Universal Robots PolyScope program: DAS428_958_10_MAR_21_DAS_lado_izquierdo.urp

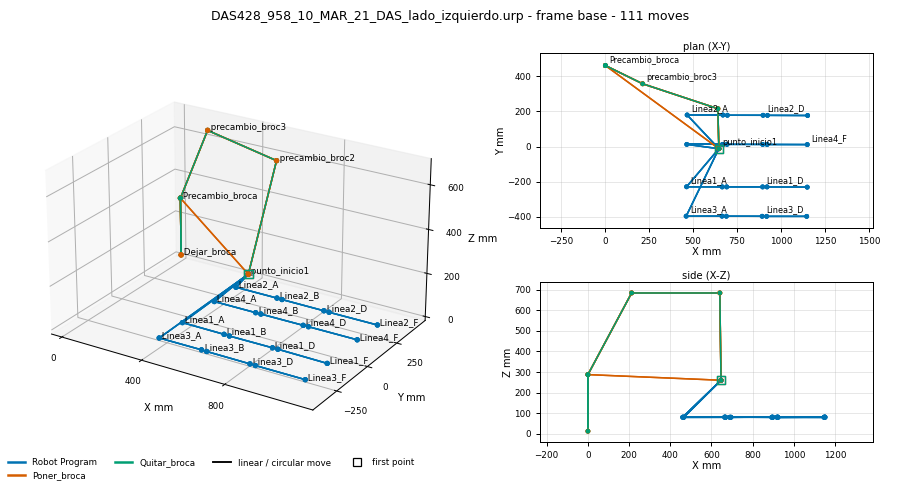
[picture p0: tool path of DAS428_958_10_MAR_21_DAS_lado_izquierdo.urp in frame base, 111 of 219 moves have a stored position in this frame; points joined in program order, loops and branches not executed]
Program DAS428_958_10_MAR_21_DAS_lado_izquierdo (installation=instalacion_derecha_10_MAR_21 directory=/programs/izquierdo createdIn=5.6.0.90886 lastSavedIn=5.6.0.90886 robotSerialNumber=20195001785)
Calibrated DH parameters: a=[0.000107, -0.568984, -0.552934, -0.00001, -0.000063, 0]; d=[0.180718, -257.998067, 200.685024, 57.48776, 0.119923, 0.115353]; alpha=[1.571119, 0.000876, -0.002498, 1.571178, -1.570523, 0]; deltaTheta=[0, -0.378191, 0.631587, -0.253396, 0, 0]
Robot Program (runOnlyOnce=false)
  Folder Variables
    bajada_broca := p[0,0,-0.008,0,0,0]
    barrenos_menos1 := 0
    barreno_actual := 0
    posicion := p[0,0,300,0,0,0]
    cambiar_broca := False
    barrenos_hechos := 0
    eje7 := 3
    Wait Sleep waitTime=0.5
  Folder Home
    Wait Sleep waitTime=0.3
    SafeHome (positionOptionType=SPEED_AND_ACCELERATION speed=1.047198 acceleration=1.396263 nextMotionTime=2)
    SuppressedNode
      MoveL speed 250 mm/s, acceleration 1200 mm/s^2 (useActiveTCP=true) feature=Base
        Waypoint home_trans: TCP in base x=-171.077 y=546.65 z=109.574 mm, rx=0.1544 ry=3.1247 rz=-0.2011 rad; joints [-91.802, -93.053, 127.954, -27.005, -275.278, -0.192] deg; TCP offset x=0.411 y=-218.298 z=37.994 mm, rx=1.558 ry=-0.1255 rz=0.1212 rad
    Wait Sleep waitTime=0.3
    iniciando_prog := True
    Call Poner_broca
  Folder Posicion2
    eje7 := 2
    Folder Broca_1
      Folder Linea1
        Folder Marcar_puntos
          MoveL speed 100 mm/s, acceleration 500 mm/s^2 (useActiveTCP=true) feature=Base
            SafeHome (positionOptionType=SPEED_AND_ACCELERATION speed=1.047198 acceleration=1.396263 nextMotionTime=2)
            Waypoint punto_inicio1: TCP in base x=646.451 y=-11.704 z=260.166 mm, rx=2.1511 ry=2.2897 rz=0 rad; joints [-205.616, -96.356, 115.768, -18.693, -308.324, -0.329] deg; TCP offset x=0.411 y=-218.298 z=37.994 mm, rx=1.558 ry=-0.1255 rz=0.1212 rad
            Waypoint Linea1_A: TCP in base x=462.97 y=-228.381 z=81.417 mm, rx=3.1274 ry=-0.0942 rz=0.0027 rad; joints [-212.166, -91.385, 132.289, -41.367, -217.89, -0.202] deg; TCP offset x=0.411 y=-218.298 z=37.994 mm, rx=1.558 ry=-0.1255 rz=0.1212 rad
            Waypoint Linea1_B: TCP in base x=665.709 y=-229.051 z=81.124 mm, rx=3.1274 ry=-0.0942 rz=0.0027 rad; joints [-202.097, -73.27, 110.874, -38.21, -207.821, -0.358] deg
            Waypoint Linea1_C: TCP in base x=691.124 y=-228.949 z=80.167 mm, rx=3.1274 ry=-0.0942 rz=0.0027 rad; joints [-201.251, -71.148, 108.001, -37.475, -206.974, -0.377] deg
            Waypoint Linea1_D: TCP in base x=895.378 y=-229.075 z=81.054 mm, rx=3.0494 ry=0.7125 rz=-0.0018 rad; joints [-199.71, -60.243, 91.126, -30.929, -235.176, -0.15] deg
            Waypoint Linea1_E: TCP in base x=920.631 y=-228.998 z=81.3 mm, rx=3.0494 ry=0.7125 rz=-0.0016 rad; joints [-199.108, -58.185, 87.734, -29.605, -234.57, -0.15] deg
            Waypoint Linea1_F: TCP in base x=1149.195 y=-230.503 z=80.116 mm, rx=3.0494 ry=0.7125 rz=-0.0018 rad; joints [-195.083, -36.259, 48.872, -12.673, -230.505, -0.164] deg
        Folder AB
          'desbaste_inicial'
          bajada_broca := p[0,0,-0.008,0,0,0]
          barrenos_menos1 := 8
          barreno_actual := 0
          Loop While (checkContinuously=false) expression=barreno_actual≤barrenos_menos1
            Folder Perforacion
              MoveL speed 100 mm/s, acceleration 500 mm/s^2 (useActiveTCP=true) feature=Base
                internos := interpolate_pose(Linea1_A, Linea1_B, barreno_actual/barrenos_menos1)
                Waypoint Waypoint (Variable): variable=internos
                'desbaste_inicial'
                bajada_broca := p[0,0,-0.008,0,0,0]
                bajada := p[0,0,0.008,0,0,0]
                MoveDirectionNode (selectedDirection=ZMinus toolParams=0.003, 0.005)
                  Until DISTANCE (allowActions=false deceleration=3 distanceNodeType=STOP) Distance=0.054; motionParameters(blendRadius=0)
                Popup Message (haltProgram=false message=punto contacto alanzdo inputType=Text)
                MoveDirectionNode (selectedDirection=ZPlus toolParams=0.003, 0.005)
                  Until DISTANCE (allowActions=false deceleration=3 distanceNodeType=STOP) Distance=0.002; motionParameters(blendRadius=0)
                Wait Sleep waitTime=0.3
                Set DigitalOutput pin=config_out[1]; digitalValue=1
                Wait Sleep waitTime=0.3
                Loop Counting (count=3) loopVariable(name=Loop_11)
                  bajar := pose_add(get_actual_tcp_pose(), bajada_broca)
                  Waypoint Waypoint (Variable): motionParameters(jointSpeed=1.047198 jointAcceleration=1.396263 cartesianSpeed=0.001 cartesianAcceleration=0.005); variable=bajar
                  subir := pose_sub(get_actual_tcp_pose(), bajada_broca)
                  Waypoint Waypoint (Variable): motionParameters(jointSpeed=1.047198 jointAcceleration=1.396263 cartesianSpeed=0.005 cartesianAcceleration=0.01); variable=subir
                  bajada_broca := pose_sub(bajada_broca, bajada)
                MoveDirectionNode (selectedDirection=ZPlus toolParams=0.03, 0.035)
                  Until DISTANCE (allowActions=false deceleration=3 distanceNodeType=STOP) Distance=0.06; motionParameters(blendRadius=0)
                Set DigitalOutput pin=config_out[1]; digitalValue=0
                barreno_actual := barreno_actual+1
                Call Quitar_broca
                Call Poner_broca
        Folder CD
          'desbaste_inicial'
          bajada_broca := p[0,0,-0.008,0,0,0]
          barrenos_menos1 := 8
          barreno_actual := 0
          Loop While (checkContinuously=false) expression=barreno_actual≤barrenos_menos1
            Folder Perforacion
              MoveL speed 100 mm/s, acceleration 500 mm/s^2 (useActiveTCP=true) feature=Base
                internos := interpolate_pose(Linea1_C, Linea1_D, barreno_actual/barrenos_menos1)
                Waypoint Waypoint (Variable): variable=internos
                'desbaste_inicial'
                bajada_broca := p[0,0,-0.008,0,0,0]
                bajada := p[0,0,0.008,0,0,0]
                MoveDirectionNode (selectedDirection=ZMinus toolParams=0.003, 0.005)
                  Until DISTANCE (allowActions=false deceleration=3 distanceNodeType=STOP) Distance=0.054; motionParameters(blendRadius=0)
                Popup Message (haltProgram=false message=punto contacto alanzdo inputType=Text)
                MoveDirectionNode (selectedDirection=ZPlus toolParams=0.003, 0.005)
                  Until DISTANCE (allowActions=false deceleration=3 distanceNodeType=STOP) Distance=0.002; motionParameters(blendRadius=0)
                Wait Sleep waitTime=0.3
                Set DigitalOutput pin=config_out[1]; digitalValue=1
                Wait Sleep waitTime=0.3
                Loop Counting (count=3) loopVariable(name=Loop_14)
                  bajar := pose_add(get_actual_tcp_pose(), bajada_broca)
                  Waypoint Waypoint (Variable): motionParameters(jointSpeed=1.047198 jointAcceleration=1.396263 cartesianSpeed=0.001 cartesianAcceleration=0.005); variable=bajar
                  subir := pose_sub(get_actual_tcp_pose(), bajada_broca)
                  Waypoint Waypoint (Variable): motionParameters(jointSpeed=1.047198 jointAcceleration=1.396263 cartesianSpeed=0.005 cartesianAcceleration=0.01); variable=subir
                  bajada_broca := pose_sub(bajada_broca, bajada)
                MoveDirectionNode (selectedDirection=ZPlus toolParams=0.03, 0.035)
                  Until DISTANCE (allowActions=false deceleration=3 distanceNodeType=STOP) Distance=0.06; motionParameters(blendRadius=0)
                Set DigitalOutput pin=config_out[1]; digitalValue=0
                barreno_actual := barreno_actual+1
                Call Quitar_broca
                Call Poner_broca
        Folder EF
          'desbaste_inicial'
          bajada_broca := p[0,0,-0.008,0,0,0]
          barrenos_menos1 := 9
          barreno_actual := 0
          Loop While (checkContinuously=false) expression=barreno_actual≤barrenos_menos1
            Folder Perforacion
              MoveL speed 100 mm/s, acceleration 500 mm/s^2 (useActiveTCP=true) feature=Base
                internos := interpolate_pose(Linea1_E, Linea1_F, barreno_actual/barrenos_menos1)
                Waypoint Waypoint (Variable): variable=internos
                'desbaste_inicial'
                bajada_broca := p[0,0,-0.008,0,0,0]
                bajada := p[0,0,0.008,0,0,0]
                MoveDirectionNode (selectedDirection=ZMinus toolParams=0.003, 0.005)
                  Until DISTANCE (allowActions=false deceleration=3 distanceNodeType=STOP) Distance=0.054; motionParameters(blendRadius=0)
                Popup Message (haltProgram=false message=punto contacto alanzdo inputType=Text)
                MoveDirectionNode (selectedDirection=ZPlus toolParams=0.003, 0.005)
                  Until DISTANCE (allowActions=false deceleration=3 distanceNodeType=STOP) Distance=0.002; motionParameters(blendRadius=0)
                Wait Sleep waitTime=0.3
                Set DigitalOutput pin=config_out[1]; digitalValue=1
                Wait Sleep waitTime=0.3
                Loop Counting (count=3) loopVariable(name=Loop_16)
                  bajar := pose_add(get_actual_tcp_pose(), bajada_broca)
                  Waypoint Waypoint (Variable): motionParameters(jointSpeed=1.047198 jointAcceleration=1.396263 cartesianSpeed=0.001 cartesianAcceleration=0.005); variable=bajar
                  subir := pose_sub(get_actual_tcp_pose(), bajada_broca)
                  Waypoint Waypoint (Variable): motionParameters(jointSpeed=1.047198 jointAcceleration=1.396263 cartesianSpeed=0.005 cartesianAcceleration=0.01); variable=subir
                  bajada_broca := pose_sub(bajada_broca, bajada)
                MoveDirectionNode (selectedDirection=ZPlus toolParams=0.03, 0.035)
                  Until DISTANCE (allowActions=false deceleration=3 distanceNodeType=STOP) Distance=0.06; motionParameters(blendRadius=0)
                Set DigitalOutput pin=config_out[1]; digitalValue=0
                barreno_actual := barreno_actual+1
                Call Quitar_broca
                Call Poner_broca
      Popup Message (haltProgram=false message=Linea1 con chica Terminada! inputType=Text)
      Folder Linea2
        Folder Marcar_puntos
          MoveL speed 100 mm/s, acceleration 500 mm/s^2 (useActiveTCP=true) feature=Base
            Waypoint punto_inicio1: TCP in base x=646.451 y=-11.704 z=260.166 mm, rx=2.1511 ry=2.2897 rz=0 rad; joints [-205.616, -96.356, 115.768, -18.693, -308.324, -0.329] deg; TCP offset x=0.411 y=-218.298 z=37.994 mm, rx=1.558 ry=-0.1255 rz=0.1212 rad
            Waypoint Linea2_A: TCP in base x=466.152 y=180.095 z=80.596 mm, rx=2.7092 ry=1.5752 rz=0.0035 rad; joints [-170.07, -97.302, 137.574, -40.225, -239.59, -0.018] deg; TCP offset x=0.411 y=-218.298 z=37.994 mm, rx=1.558 ry=-0.1255 rz=0.1212 rad
            Waypoint Linea2_B: TCP in base x=669.642 y=179.866 z=80.737 mm, rx=2.7092 ry=1.5752 rz=0.0035 rad; joints [-173.706, -79.789, 119.419, -39.574, -243.231, -0.007] deg
            Waypoint Linea2_C: TCP in base x=694.939 y=178.643 z=80.843 mm, rx=2.7092 ry=1.5752 rz=0.0035 rad; joints [-174.103, -77.842, 116.933, -39.035, -243.627, -0.006] deg
            Waypoint Linea2_D: TCP in base x=897.97 y=178.427 z=80.373 mm, rx=2.7092 ry=1.5752 rz=0.0035 rad; joints [-175.658, -62.16, 94.258, -32.04, -245.171, -0.008] deg
            Waypoint Linea2_E: TCP in base x=923.127 y=178.076 z=79.947 mm, rx=2.7092 ry=1.5752 rz=0.0035 rad; joints [-175.819, -60.176, 91.121, -30.888, -245.33, -0.008] deg
            Waypoint Linea2_F: TCP in base x=1151.498 y=177.179 z=80.752 mm, rx=2.7092 ry=1.5752 rz=0.0035 rad; joints [-176.803, -39.928, 55.644, -15.661, -246.279, -0.017] deg
        Folder AB
          'desbaste_inicial'
          bajada_broca := p[0,0,-0.008,0,0,0]
          barrenos_menos1 := 8
          barreno_actual := 0
          Loop While (checkContinuously=false) expression=barreno_actual≤barrenos_menos1
            Folder Perforacion
              MoveL speed 100 mm/s, acceleration 500 mm/s^2 (useActiveTCP=true) feature=Base
                internos := interpolate_pose(Linea2_A, Linea2_B, barreno_actual/barrenos_menos1)
                Waypoint Waypoint (Variable): variable=internos
                'desbaste_inicial'
                bajada_broca := p[0,0,-0.008,0,0,0]
                bajada := p[0,0,0.008,0,0,0]
                MoveDirectionNode (selectedDirection=ZMinus toolParams=0.003, 0.005)
                  Until DISTANCE (allowActions=false deceleration=3 distanceNodeType=STOP) Distance=0.054; motionParameters(blendRadius=0)
                Popup Message (haltProgram=false message=punto contacto alanzdo inputType=Text)
                MoveDirectionNode (selectedDirection=ZPlus toolParams=0.003, 0.005)
                  Until DISTANCE (allowActions=false deceleration=3 distanceNodeType=STOP) Distance=0.002; motionParameters(blendRadius=0)
                Wait Sleep waitTime=0.3
                Set DigitalOutput pin=config_out[1]; digitalValue=1
                Wait Sleep waitTime=0.3
                Loop Counting (count=3) loopVariable(name=Loop_2)
                  bajar := pose_add(get_actual_tcp_pose(), bajada_broca)
                  Waypoint Waypoint (Variable): motionParameters(jointSpeed=1.047198 jointAcceleration=1.396263 cartesianSpeed=0.001 cartesianAcceleration=0.005); variable=bajar
                  subir := pose_sub(get_actual_tcp_pose(), bajada_broca)
                  Waypoint Waypoint (Variable): motionParameters(jointSpeed=1.047198 jointAcceleration=1.396263 cartesianSpeed=0.005 cartesianAcceleration=0.01); variable=subir
                  bajada_broca := pose_sub(bajada_broca, bajada)
                MoveDirectionNode (selectedDirection=ZPlus toolParams=0.03, 0.035)
                  Until DISTANCE (allowActions=false deceleration=3 distanceNodeType=STOP) Distance=0.06; motionParameters(blendRadius=0)
                Set DigitalOutput pin=config_out[1]; digitalValue=0
                barreno_actual := barreno_actual+1
                Call Quitar_broca
                Call Poner_broca
        Folder CD
          'desbaste_inicial'
          bajada_broca := p[0,0,-0.008,0,0,0]
          barrenos_menos1 := 8
          barreno_actual := 0
          Loop While (checkContinuously=false) expression=barreno_actual≤barrenos_menos1
            Folder Perforacion
              MoveL speed 100 mm/s, acceleration 500 mm/s^2 (useActiveTCP=true) feature=Base
                internos := interpolate_pose(Linea2_C, Linea2_D, barreno_actual/barrenos_menos1)
                Waypoint Waypoint (Variable): variable=internos
                'desbaste_inicial'
                bajada_broca := p[0,0,-0.008,0,0,0]
                bajada := p[0,0,0.008,0,0,0]
                MoveDirectionNode (selectedDirection=ZMinus toolParams=0.003, 0.005)
                  Until DISTANCE (allowActions=false deceleration=3 distanceNodeType=STOP) Distance=0.054; motionParameters(blendRadius=0)
                Popup Message (haltProgram=false message=punto contacto alanzdo inputType=Text)
                MoveDirectionNode (selectedDirection=ZPlus toolParams=0.003, 0.005)
                  Until DISTANCE (allowActions=false deceleration=3 distanceNodeType=STOP) Distance=0.002; motionParameters(blendRadius=0)
                Wait Sleep waitTime=0.3
                Set DigitalOutput pin=config_out[1]; digitalValue=1
                Wait Sleep waitTime=0.3
                Loop Counting (count=3) loopVariable(name=Loop_5)
                  bajar := pose_add(get_actual_tcp_pose(), bajada_broca)
                  Waypoint Waypoint (Variable): motionParameters(jointSpeed=1.047198 jointAcceleration=1.396263 cartesianSpeed=0.001 cartesianAcceleration=0.005); variable=bajar
                  subir := pose_sub(get_actual_tcp_pose(), bajada_broca)
                  Waypoint Waypoint (Variable): motionParameters(jointSpeed=1.047198 jointAcceleration=1.396263 cartesianSpeed=0.005 cartesianAcceleration=0.01); variable=subir
                  bajada_broca := pose_sub(bajada_broca, bajada)
                MoveDirectionNode (selectedDirection=ZPlus toolParams=0.03, 0.035)
                  Until DISTANCE (allowActions=false deceleration=3 distanceNodeType=STOP) Distance=0.06; motionParameters(blendRadius=0)
                Set DigitalOutput pin=config_out[1]; digitalValue=0
                barreno_actual := barreno_actual+1
                Call Quitar_broca
                Call Poner_broca
        Folder EF
          'desbaste_inicial'
          bajada_broca := p[0,0,-0.008,0,0,0]
          barrenos_menos1 := 9
          barreno_actual := 0
          Loop While (checkContinuously=false) expression=barreno_actual≤barrenos_menos1
            Folder Perforacion
              MoveL speed 100 mm/s, acceleration 500 mm/s^2 (useActiveTCP=true) feature=Base
                internos := interpolate_pose(Linea2_E, Linea2_F, barreno_actual/barrenos_menos1)
                Waypoint Waypoint (Variable): variable=internos
                'desbaste_inicial'
                bajada_broca := p[0,0,-0.008,0,0,0]
                bajada := p[0,0,0.008,0,0,0]
                MoveDirectionNode (selectedDirection=ZMinus toolParams=0.003, 0.005)
                  Until DISTANCE (allowActions=false deceleration=3 distanceNodeType=STOP) Distance=0.054; motionParameters(blendRadius=0)
                Popup Message (haltProgram=false message=punto contacto alanzdo inputType=Text)
                MoveDirectionNode (selectedDirection=ZPlus toolParams=0.003, 0.005)
                  Until DISTANCE (allowActions=false deceleration=3 distanceNodeType=STOP) Distance=0.002; motionParameters(blendRadius=0)
                Wait Sleep waitTime=0.3
                Set DigitalOutput pin=config_out[1]; digitalValue=1
                Wait Sleep waitTime=0.3
                Loop Counting (count=3) loopVariable(name=Loop_9)
                  bajar := pose_add(get_actual_tcp_pose(), bajada_broca)
                  Waypoint Waypoint (Variable): motionParameters(jointSpeed=1.047198 jointAcceleration=1.396263 cartesianSpeed=0.001 cartesianAcceleration=0.005); variable=bajar
                  subir := pose_sub(get_actual_tcp_pose(), bajada_broca)
                  Waypoint Waypoint (Variable): motionParameters(jointSpeed=1.047198 jointAcceleration=1.396263 cartesianSpeed=0.005 cartesianAcceleration=0.01); variable=subir
                  bajada_broca := pose_sub(bajada_broca, bajada)
                MoveDirectionNode (selectedDirection=ZPlus toolParams=0.03, 0.035)
                  Until DISTANCE (allowActions=false deceleration=3 distanceNodeType=STOP) Distance=0.06; motionParameters(blendRadius=0)
                Set DigitalOutput pin=config_out[1]; digitalValue=0
                barreno_actual := barreno_actual+1
                If barreno_actual>barrenos_menos1
                  cambiar_broca := True
                Call Quitar_broca
                Call Poner_broca
      Popup Message (haltProgram=false message=Linea2 con chica Terminada! inputType=Text)
    Folder Broca_2
      Folder Linea1
        Folder Marcar_puntos
          MoveL speed 100 mm/s, acceleration 500 mm/s^2 (useActiveTCP=true) feature=Base
            Waypoint punto_inicio1: TCP in base x=646.451 y=-11.704 z=260.166 mm, rx=2.1511 ry=2.2897 rz=0 rad; joints [-205.616, -96.356, 115.768, -18.693, -308.324, -0.329] deg; TCP offset x=0.411 y=-218.298 z=37.994 mm, rx=1.558 ry=-0.1255 rz=0.1212 rad
            Waypoint Linea1_A: TCP in base x=462.97 y=-228.381 z=81.417 mm, rx=3.1274 ry=-0.0942 rz=0.0027 rad; joints [-212.166, -91.385, 132.289, -41.367, -217.89, -0.202] deg; TCP offset x=0.411 y=-218.298 z=37.994 mm, rx=1.558 ry=-0.1255 rz=0.1212 rad
            Waypoint Linea1_B: TCP in base x=665.709 y=-229.051 z=81.124 mm, rx=3.1274 ry=-0.0942 rz=0.0027 rad; joints [-202.097, -73.27, 110.874, -38.21, -207.821, -0.358] deg
            Waypoint Linea1_C: TCP in base x=691.124 y=-228.949 z=80.167 mm, rx=3.1274 ry=-0.0942 rz=0.0027 rad; joints [-201.251, -71.148, 108.001, -37.475, -206.974, -0.377] deg
            Waypoint Linea1_D: TCP in base x=895.378 y=-229.075 z=81.054 mm, rx=3.0494 ry=0.7125 rz=-0.0018 rad; joints [-199.71, -60.243, 91.126, -30.929, -235.176, -0.15] deg
            Waypoint Linea1_E: TCP in base x=920.631 y=-228.998 z=81.3 mm, rx=3.0494 ry=0.7125 rz=-0.0016 rad; joints [-199.108, -58.185, 87.734, -29.605, -234.57, -0.15] deg
            Waypoint Linea1_F: TCP in base x=1149.195 y=-230.503 z=80.116 mm, rx=3.0494 ry=0.7125 rz=-0.0018 rad; joints [-195.083, -36.259, 48.872, -12.673, -230.505, -0.164] deg
        Folder AB
          'desbaste_inicial'
          bajada_broca := p[0,0,-0.012,0,0,0]
          barrenos_menos1 := 8
          barreno_actual := 0
          Loop While (checkContinuously=false) expression=barreno_actual≤barrenos_menos1
            Folder Perforacion
              MoveL speed 100 mm/s, acceleration 500 mm/s^2 (useActiveTCP=true) feature=Base
                internos := interpolate_pose(Linea1_A, Linea1_B, barreno_actual/barrenos_menos1)
                Waypoint Waypoint (Variable): variable=internos
                'desbaste_inicial'
                bajada_broca := p[0,0,-0.012,0,0,0]
                bajada := p[0,0,0.012,0,0,0]
                MoveDirectionNode (selectedDirection=ZMinus toolParams=0.01, 0.015)
                  Until DISTANCE (allowActions=false deceleration=3 distanceNodeType=STOP) Distance=0.054; motionParameters(blendRadius=0)
                Popup Message (haltProgram=false message=punto contacto alanzdo inputType=Text)
                MoveDirectionNode (selectedDirection=ZPlus toolParams=0.003, 0.005)
                  Until DISTANCE (allowActions=false deceleration=3 distanceNodeType=STOP) Distance=0.002; motionParameters(blendRadius=0)
                Wait Sleep waitTime=0.3
                Set DigitalOutput pin=config_out[1]; digitalValue=1
                Wait Sleep waitTime=0.3
                Loop Counting (count=2) loopVariable(name=Loop_46)
                  bajar := pose_add(get_actual_tcp_pose(), bajada_broca)
                  Waypoint Waypoint (Variable): motionParameters(jointSpeed=1.047198 jointAcceleration=1.396263 cartesianSpeed=0.001 cartesianAcceleration=0.005); variable=bajar
                  subir := pose_sub(get_actual_tcp_pose(), bajada_broca)
                  Waypoint Waypoint (Variable): motionParameters(jointSpeed=1.047198 jointAcceleration=1.396263 cartesianSpeed=0.005 cartesianAcceleration=0.01); variable=subir
                  bajada_broca := pose_sub(bajada_broca, bajada)
                MoveDirectionNode (selectedDirection=ZPlus toolParams=0.03, 0.035)
                  Until DISTANCE (allowActions=false deceleration=3 distanceNodeType=STOP) Distance=0.06; motionParameters(blendRadius=0)
                Set DigitalOutput pin=config_out[1]; digitalValue=0
                barreno_actual := barreno_actual+1
                Call Quitar_broca
                Call Poner_broca
        Folder CD
          'desbaste_inicial'
          bajada_broca := p[0,0,-0.012,0,0,0]
          barrenos_menos1 := 8
          barreno_actual := 0
          Loop While (checkContinuously=false) expression=barreno_actual≤barrenos_menos1
            Folder Perforacion
              MoveL speed 100 mm/s, acceleration 500 mm/s^2 (useActiveTCP=true) feature=Base
                internos := interpolate_pose(Linea1_C, Linea1_D, barreno_actual/barrenos_menos1)
                Waypoint Waypoint (Variable): variable=internos
                'desbaste_inicial'
                bajada_broca := p[0,0,-0.012,0,0,0]
                bajada := p[0,0,0.012,0,0,0]
                MoveDirectionNode (selectedDirection=ZMinus toolParams=0.01, 0.015)
                  Until DISTANCE (allowActions=false deceleration=3 distanceNodeType=STOP) Distance=0.054; motionParameters(blendRadius=0)
                Popup Message (haltProgram=false message=punto contacto alanzdo inputType=Text)
                MoveDirectionNode (selectedDirection=ZPlus toolParams=0.003, 0.005)
                  Until DISTANCE (allowActions=false deceleration=3 distanceNodeType=STOP) Distance=0.002; motionParameters(blendRadius=0)
                Wait Sleep waitTime=0.3
                Set DigitalOutput pin=config_out[1]; digitalValue=1
                Wait Sleep waitTime=0.3
                Loop Counting (count=2) loopVariable(name=Loop_48)
                  bajar := pose_add(get_actual_tcp_pose(), bajada_broca)
                  Waypoint Waypoint (Variable): motionParameters(jointSpeed=1.047198 jointAcceleration=1.396263 cartesianSpeed=0.001 cartesianAcceleration=0.005); variable=bajar
                  subir := pose_sub(get_actual_tcp_pose(), bajada_broca)
                  Waypoint Waypoint (Variable): motionParameters(jointSpeed=1.047198 jointAcceleration=1.396263 cartesianSpeed=0.005 cartesianAcceleration=0.01); variable=subir
                  bajada_broca := pose_sub(bajada_broca, bajada)
                MoveDirectionNode (selectedDirection=ZPlus toolParams=0.03, 0.035)
                  Until DISTANCE (allowActions=false deceleration=3 distanceNodeType=STOP) Distance=0.06; motionParameters(blendRadius=0)
                Set DigitalOutput pin=config_out[1]; digitalValue=0
                barreno_actual := barreno_actual+1
                Call Quitar_broca
                Call Poner_broca
        Folder EF
          'desbaste_inicial'
          bajada_broca := p[0,0,-0.012,0,0,0]
          barrenos_menos1 := 9
          barreno_actual := 0
          Loop While (checkContinuously=false) expression=barreno_actual≤barrenos_menos1
            Folder Perforacion
              MoveL speed 100 mm/s, acceleration 500 mm/s^2 (useActiveTCP=true) feature=Base
                internos := interpolate_pose(Linea1_E, Linea1_F, barreno_actual/barrenos_menos1)
                Waypoint Waypoint (Variable): variable=internos
                'desbaste_inicial'
                bajada_broca := p[0,0,-0.012,0,0,0]
                bajada := p[0,0,0.012,0,0,0]
                MoveDirectionNode (selectedDirection=ZMinus toolParams=0.01, 0.015)
                  Until DISTANCE (allowActions=false deceleration=3 distanceNodeType=STOP) Distance=0.054; motionParameters(blendRadius=0)
                Popup Message (haltProgram=false message=punto contacto alanzdo inputType=Text)
                MoveDirectionNode (selectedDirection=ZPlus toolParams=0.003, 0.005)
                  Until DISTANCE (allowActions=false deceleration=3 distanceNodeType=STOP) Distance=0.002; motionParameters(blendRadius=0)
                Wait Sleep waitTime=0.3
                Set DigitalOutput pin=config_out[1]; digitalValue=1
                Wait Sleep waitTime=0.3
                Loop Counting (count=2) loopVariable(name=Loop_50)
                  bajar := pose_add(get_actual_tcp_pose(), bajada_broca)
                  Waypoint Waypoint (Variable): motionParameters(jointSpeed=1.047198 jointAcceleration=1.396263 cartesianSpeed=0.001 cartesianAcceleration=0.005); variable=bajar
                  subir := pose_sub(get_actual_tcp_pose(), bajada_broca)
                  Waypoint Waypoint (Variable): motionParameters(jointSpeed=1.047198 jointAcceleration=1.396263 cartesianSpeed=0.005 cartesianAcceleration=0.01); variable=subir
                  bajada_broca := pose_sub(bajada_broca, bajada)
                MoveDirectionNode (selectedDirection=ZPlus toolParams=0.03, 0.035)
                  Until DISTANCE (allowActions=false deceleration=3 distanceNodeType=STOP) Distance=0.06; motionParameters(blendRadius=0)
                Set DigitalOutput pin=config_out[1]; digitalValue=0
                barreno_actual := barreno_actual+1
                Call Quitar_broca
                Call Poner_broca
      Popup Message (haltProgram=false message=Linea1 con media Terminada! inputType=Text)
      Folder Linea2
        Folder Marcar_puntos
          MoveL speed 100 mm/s, acceleration 500 mm/s^2 (useActiveTCP=true) feature=Base
            Waypoint punto_inicio1: TCP in base x=646.451 y=-11.704 z=260.166 mm, rx=2.1511 ry=2.2897 rz=0 rad; joints [-205.616, -96.356, 115.768, -18.693, -308.324, -0.329] deg; TCP offset x=0.411 y=-218.298 z=37.994 mm, rx=1.558 ry=-0.1255 rz=0.1212 rad
            Waypoint Linea2_A: TCP in base x=466.152 y=180.095 z=80.596 mm, rx=2.7092 ry=1.5752 rz=0.0035 rad; joints [-170.07, -97.302, 137.574, -40.225, -239.59, -0.018] deg; TCP offset x=0.411 y=-218.298 z=37.994 mm, rx=1.558 ry=-0.1255 rz=0.1212 rad
            Waypoint Linea2_B: TCP in base x=669.642 y=179.866 z=80.737 mm, rx=2.7092 ry=1.5752 rz=0.0035 rad; joints [-173.706, -79.789, 119.419, -39.574, -243.231, -0.007] deg
            Waypoint Linea2_C: TCP in base x=694.939 y=178.643 z=80.843 mm, rx=2.7092 ry=1.5752 rz=0.0035 rad; joints [-174.103, -77.842, 116.933, -39.035, -243.627, -0.006] deg
            Waypoint Linea2_D: TCP in base x=897.97 y=178.427 z=80.373 mm, rx=2.7092 ry=1.5752 rz=0.0035 rad; joints [-175.658, -62.16, 94.258, -32.04, -245.171, -0.008] deg
            Waypoint Linea2_E: TCP in base x=923.127 y=178.076 z=79.947 mm, rx=2.7092 ry=1.5752 rz=0.0035 rad; joints [-175.819, -60.176, 91.121, -30.888, -245.33, -0.008] deg
            Waypoint Linea2_F: TCP in base x=1151.498 y=177.179 z=80.752 mm, rx=2.7092 ry=1.5752 rz=0.0035 rad; joints [-176.803, -39.928, 55.644, -15.661, -246.279, -0.017] deg
        Folder AB
          'desbaste_inicial'
          bajada_broca := p[0,0,-0.012,0,0,0]
          barrenos_menos1 := 8
          barreno_actual := 0
          Loop While (checkContinuously=false) expression=barreno_actual≤barrenos_menos1
            Folder Perforacion
              MoveL speed 100 mm/s, acceleration 500 mm/s^2 (useActiveTCP=true) feature=Base
                internos := interpolate_pose(Linea2_A, Linea2_B, barreno_actual/barrenos_menos1)
                Waypoint Waypoint (Variable): variable=internos
                'desbaste_inicial'
                bajada_broca := p[0,0,-0.012,0,0,0]
                bajada := p[0,0,0.012,0,0,0]
                MoveDirectionNode (selectedDirection=ZMinus toolParams=0.02, 0.015)
                  Until DISTANCE (allowActions=false deceleration=3 distanceNodeType=STOP) Distance=0.054; motionParameters(blendRadius=0)
                Popup Message (haltProgram=false message=punto contacto alanzdo inputType=Text)
                MoveDirectionNode (selectedDirection=ZPlus toolParams=0.003, 0.005)
                  Until DISTANCE (allowActions=false deceleration=3 distanceNodeType=STOP) Distance=0.002; motionParameters(blendRadius=0)
                Wait Sleep waitTime=0.3
                Set DigitalOutput pin=config_out[1]; digitalValue=1
                Wait Sleep waitTime=0.3
                Loop Counting (count=2) loopVariable(name=Loop_34)
                  bajar := pose_add(get_actual_tcp_pose(), bajada_broca)
                  Waypoint Waypoint (Variable): motionParameters(jointSpeed=1.047198 jointAcceleration=1.396263 cartesianSpeed=0.001 cartesianAcceleration=0.005); variable=bajar
                  subir := pose_sub(get_actual_tcp_pose(), bajada_broca)
                  Waypoint Waypoint (Variable): motionParameters(jointSpeed=1.047198 jointAcceleration=1.396263 cartesianSpeed=0.005 cartesianAcceleration=0.01); variable=subir
                  bajada_broca := pose_sub(bajada_broca, bajada)
                MoveDirectionNode (selectedDirection=ZPlus toolParams=0.03, 0.035)
                  Until DISTANCE (allowActions=false deceleration=3 distanceNodeType=STOP) Distance=0.06; motionParameters(blendRadius=0)
                Set DigitalOutput pin=config_out[1]; digitalValue=0
                barreno_actual := barreno_actual+1
                Call Quitar_broca
                Call Poner_broca
        Folder CD
          'desbaste_inicial'
          bajada_broca := p[0,0,-0.012,0,0,0]
          barrenos_menos1 := 8
          barreno_actual := 0
          Loop While (checkContinuously=false) expression=barreno_actual≤barrenos_menos1
            Folder Perforacion
              MoveL speed 100 mm/s, acceleration 500 mm/s^2 (useActiveTCP=true) feature=Base
                internos := interpolate_pose(Linea2_C, Linea2_D, barreno_actual/barrenos_menos1)
                Waypoint Waypoint (Variable): variable=internos
                'desbaste_inicial'
                bajada_broca := p[0,0,-0.012,0,0,0]
                bajada := p[0,0,0.012,0,0,0]
                MoveDirectionNode (selectedDirection=ZMinus toolParams=0.02, 0.015)
                  Until DISTANCE (allowActions=false deceleration=3 distanceNodeType=STOP) Distance=0.054; motionParameters(blendRadius=0)
                Popup Message (haltProgram=false message=punto contacto alanzdo inputType=Text)
                MoveDirectionNode (selectedDirection=ZPlus toolParams=0.003, 0.005)
                  Until DISTANCE (allowActions=false deceleration=3 distanceNodeType=STOP) Distance=0.002; motionParameters(blendRadius=0)
                Wait Sleep waitTime=0.3
                Set DigitalOutput pin=config_out[1]; digitalValue=1
                Wait Sleep waitTime=0.3
                Loop Counting (count=2) loopVariable(name=Loop_36)
                  bajar := pose_add(get_actual_tcp_pose(), bajada_broca)
                  Waypoint Waypoint (Variable): motionParameters(jointSpeed=1.047198 jointAcceleration=1.396263 cartesianSpeed=0.001 cartesianAcceleration=0.005); variable=bajar
                  subir := pose_sub(get_actual_tcp_pose(), bajada_broca)
                  Waypoint Waypoint (Variable): motionParameters(jointSpeed=1.047198 jointAcceleration=1.396263 cartesianSpeed=0.005 cartesianAcceleration=0.01); variable=subir
                  bajada_broca := pose_sub(bajada_broca, bajada)
                MoveDirectionNode (selectedDirection=ZPlus toolParams=0.03, 0.035)
                  Until DISTANCE (allowActions=false deceleration=3 distanceNodeType=STOP) Distance=0.06; motionParameters(blendRadius=0)
                Set DigitalOutput pin=config_out[1]; digitalValue=0
                barreno_actual := barreno_actual+1
                Call Quitar_broca
                Call Poner_broca
        Folder EF
          'desbaste_inicial'
          bajada_broca := p[0,0,-0.012,0,0,0]
          barrenos_menos1 := 9
          barreno_actual := 0
          Loop While (checkContinuously=false) expression=barreno_actual≤barrenos_menos1
            Folder Perforacion
              MoveL speed 100 mm/s, acceleration 500 mm/s^2 (useActiveTCP=true) feature=Base
                internos := interpolate_pose(Linea2_E, Linea2_F, barreno_actual/barrenos_menos1)
                Waypoint Waypoint (Variable): variable=internos
                'desbaste_inicial'
                bajada_broca := p[0,0,-0.012,0,0,0]
                bajada := p[0,0,0.012,0,0,0]
                MoveDirectionNode (selectedDirection=ZMinus toolParams=0.02, 0.015)
                  Until DISTANCE (allowActions=false deceleration=3 distanceNodeType=STOP) Distance=0.054; motionParameters(blendRadius=0)
                Popup Message (haltProgram=false message=punto contacto alanzdo inputType=Text)
                MoveDirectionNode (selectedDirection=ZPlus toolParams=0.003, 0.005)
                  Until DISTANCE (allowActions=false deceleration=3 distanceNodeType=STOP) Distance=0.002; motionParameters(blendRadius=0)
                Wait Sleep waitTime=0.3
                Set DigitalOutput pin=config_out[1]; digitalValue=1
                Wait Sleep waitTime=0.3
                Loop Counting (count=2) loopVariable(name=Loop_38)
                  bajar := pose_add(get_actual_tcp_pose(), bajada_broca)
                  Waypoint Waypoint (Variable): motionParameters(jointSpeed=1.047198 jointAcceleration=1.396263 cartesianSpeed=0.001 cartesianAcceleration=0.005); variable=bajar
                  subir := pose_sub(get_actual_tcp_pose(), bajada_broca)
                  Waypoint Waypoint (Variable): motionParameters(jointSpeed=1.047198 jointAcceleration=1.396263 cartesianSpeed=0.005 cartesianAcceleration=0.01); variable=subir
                  bajada_broca := pose_sub(bajada_broca, bajada)
                MoveDirectionNode (selectedDirection=ZPlus toolParams=0.03, 0.035)
                  Until DISTANCE (allowActions=false deceleration=3 distanceNodeType=STOP) Distance=0.06; motionParameters(blendRadius=0)
                Set DigitalOutput pin=config_out[1]; digitalValue=0
                barreno_actual := barreno_actual+1
                If barreno_actual>barrenos_menos1
                  cambiar_broca := True
                Call Quitar_broca
                Call Poner_broca
      Popup Message (haltProgram=false message=Linea2 con media Terminada! inputType=Text)
    Folder Broca_3
      Folder Linea1
        Folder Marcar_puntos
          MoveL speed 100 mm/s, acceleration 500 mm/s^2 (useActiveTCP=true) feature=Base
            Waypoint punto_inicio1: TCP in base x=646.451 y=-11.704 z=260.166 mm, rx=2.1511 ry=2.2897 rz=0 rad; joints [-205.616, -96.356, 115.768, -18.693, -308.324, -0.329] deg; TCP offset x=0.411 y=-218.298 z=37.994 mm, rx=1.558 ry=-0.1255 rz=0.1212 rad
            Waypoint Linea1_A: TCP in base x=462.97 y=-228.381 z=81.417 mm, rx=3.1274 ry=-0.0942 rz=0.0027 rad; joints [-212.166, -91.385, 132.289, -41.367, -217.89, -0.202] deg; TCP offset x=0.411 y=-218.298 z=37.994 mm, rx=1.558 ry=-0.1255 rz=0.1212 rad
            Waypoint Linea1_B: TCP in base x=665.709 y=-229.051 z=81.124 mm, rx=3.1274 ry=-0.0942 rz=0.0027 rad; joints [-202.097, -73.27, 110.874, -38.21, -207.821, -0.358] deg
            Waypoint Linea1_C: TCP in base x=691.124 y=-228.949 z=80.167 mm, rx=3.1274 ry=-0.0942 rz=0.0027 rad; joints [-201.251, -71.148, 108.001, -37.475, -206.974, -0.377] deg
            Waypoint Linea1_D: TCP in base x=895.378 y=-229.075 z=81.054 mm, rx=3.0494 ry=0.7125 rz=-0.0018 rad; joints [-199.71, -60.243, 91.126, -30.929, -235.176, -0.15] deg
            Waypoint Linea1_E: TCP in base x=920.631 y=-228.998 z=81.3 mm, rx=3.0494 ry=0.7125 rz=-0.0016 rad; joints [-199.108, -58.185, 87.734, -29.605, -234.57, -0.15] deg
            Waypoint Linea1_F: TCP in base x=1149.195 y=-230.503 z=80.116 mm, rx=3.0494 ry=0.7125 rz=-0.0018 rad; joints [-195.083, -36.259, 48.872, -12.673, -230.505, -0.164] deg
        Folder AB
          'desbaste_inicial'
          bajada_broca := p[0,0,-0.012,0,0,0]
          barrenos_menos1 := 8
          barreno_actual := 0
          Loop While (checkContinuously=false) expression=barreno_actual≤barrenos_menos1
            Folder Perforacion
              MoveL speed 100 mm/s, acceleration 500 mm/s^2 (useActiveTCP=true) feature=Base
                internos := interpolate_pose(Linea1_A, Linea1_B, barreno_actual/barrenos_menos1)
                Waypoint Waypoint (Variable): variable=internos
                'desbaste_inicial'
                bajada_broca := p[0,0,-0.012,0,0,0]
                bajada := p[0,0,0.012,0,0,0]
                MoveDirectionNode (selectedDirection=ZMinus toolParams=0.02, 0.015)
                  Until DISTANCE (allowActions=false deceleration=3 distanceNodeType=STOP) Distance=0.055; motionParameters(blendRadius=0)
                Popup Message (haltProgram=false message=punto contacto alanzdo inputType=Text)
                MoveDirectionNode (selectedDirection=ZPlus toolParams=0.003, 0.005)
                  Until DISTANCE (allowActions=false deceleration=3 distanceNodeType=STOP) Distance=0.001; motionParameters(blendRadius=0)
                Wait Sleep waitTime=0.3
                Set DigitalOutput pin=config_out[1]; digitalValue=1
                Wait Sleep waitTime=0.3
                Loop Counting (count=2) loopVariable(name=Loop_18)
                  bajar := pose_add(get_actual_tcp_pose(), bajada_broca)
                  Waypoint Waypoint (Variable): motionParameters(jointSpeed=1.047198 jointAcceleration=1.396263 cartesianSpeed=0.001 cartesianAcceleration=0.005); variable=bajar
                  subir := pose_sub(get_actual_tcp_pose(), bajada_broca)
                  Waypoint Waypoint (Variable): motionParameters(jointSpeed=1.047198 jointAcceleration=1.396263 cartesianSpeed=0.005 cartesianAcceleration=0.01); variable=subir
                  bajada_broca := pose_sub(bajada_broca, bajada)
                MoveDirectionNode (selectedDirection=ZPlus toolParams=0.03, 0.035)
                  Until DISTANCE (allowActions=false deceleration=3 distanceNodeType=STOP) Distance=0.06; motionParameters(blendRadius=0)
                Set DigitalOutput pin=config_out[1]; digitalValue=0
                barreno_actual := barreno_actual+1
                Call Quitar_broca
                Call Poner_broca
        Folder CD
          'desbaste_inicial'
          bajada_broca := p[0,0,-0.012,0,0,0]
          barrenos_menos1 := 8
          barreno_actual := 0
          Loop While (checkContinuously=false) expression=barreno_actual≤barrenos_menos1
            Folder Perforacion
              MoveL speed 100 mm/s, acceleration 500 mm/s^2 (useActiveTCP=true) feature=Base
                internos := interpolate_pose(Linea1_C, Linea1_D, barreno_actual/barrenos_menos1)
                Waypoint Waypoint (Variable): variable=internos
                'desbaste_inicial'
                bajada_broca := p[0,0,-0.012,0,0,0]
                bajada := p[0,0,0.012,0,0,0]
                MoveDirectionNode (selectedDirection=ZMinus toolParams=0.02, 0.015)
                  Until DISTANCE (allowActions=false deceleration=3 distanceNodeType=STOP) Distance=0.055; motionParameters(blendRadius=0)
                Popup Message (haltProgram=false message=punto contacto alanzdo inputType=Text)
                MoveDirectionNode (selectedDirection=ZPlus toolParams=0.003, 0.005)
                  Until DISTANCE (allowActions=false deceleration=3 distanceNodeType=STOP) Distance=0.001; motionParameters(blendRadius=0)
                Wait Sleep waitTime=0.3
                Set DigitalOutput pin=config_out[1]; digitalValue=1
                Wait Sleep waitTime=0.3
                Loop Counting (count=2) loopVariable(name=Loop_20)
                  bajar := pose_add(get_actual_tcp_pose(), bajada_broca)
                  Waypoint Waypoint (Variable): motionParameters(jointSpeed=1.047198 jointAcceleration=1.396263 cartesianSpeed=0.001 cartesianAcceleration=0.005); variable=bajar
                  subir := pose_sub(get_actual_tcp_pose(), bajada_broca)
                  Waypoint Waypoint (Variable): motionParameters(jointSpeed=1.047198 jointAcceleration=1.396263 cartesianSpeed=0.005 cartesianAcceleration=0.01); variable=subir
                  bajada_broca := pose_sub(bajada_broca, bajada)
                MoveDirectionNode (selectedDirection=ZPlus toolParams=0.03, 0.035)
                  Until DISTANCE (allowActions=false deceleration=3 distanceNodeType=STOP) Distance=0.06; motionParameters(blendRadius=0)
                Set DigitalOutput pin=config_out[1]; digitalValue=0
                barreno_actual := barreno_actual+1
                Call Quitar_broca
                Call Poner_broca
        Folder EF
          'desbaste_inicial'
          bajada_broca := p[0,0,-0.012,0,0,0]
          barrenos_menos1 := 9
          barreno_actual := 0
          Loop While (checkContinuously=false) expression=barreno_actual≤barrenos_menos1
            Folder Perforacion
              MoveL speed 100 mm/s, acceleration 500 mm/s^2 (useActiveTCP=true) feature=Base
                internos := interpolate_pose(Linea1_E, Linea1_F, barreno_actual/barrenos_menos1)
                Waypoint Waypoint (Variable): variable=internos
                'desbaste_inicial'
                bajada_broca := p[0,0,-0.012,0,0,0]
                bajada := p[0,0,0.012,0,0,0]
                MoveDirectionNode (selectedDirection=ZMinus toolParams=0.02, 0.015)
                  Until DISTANCE (allowActions=false deceleration=3 distanceNodeType=STOP) Distance=0.055; motionParameters(blendRadius=0)
                Popup Message (haltProgram=false message=punto contacto alanzdo inputType=Text)
                MoveDirectionNode (selectedDirection=ZPlus toolParams=0.003, 0.005)
                  Until DISTANCE (allowActions=false deceleration=3 distanceNodeType=STOP) Distance=0.001; motionParameters(blendRadius=0)
                Wait Sleep waitTime=0.3
                Set DigitalOutput pin=config_out[1]; digitalValue=1
                Wait Sleep waitTime=0.3
                Loop Counting (count=2) loopVariable(name=Loop_22)
                  bajar := pose_add(get_actual_tcp_pose(), bajada_broca)
                  Waypoint Waypoint (Variable): motionParameters(jointSpeed=1.047198 jointAcceleration=1.396263 cartesianSpeed=0.001 cartesianAcceleration=0.005); variable=bajar
                  subir := pose_sub(get_actual_tcp_pose(), bajada_broca)
                  Waypoint Waypoint (Variable): motionParameters(jointSpeed=1.047198 jointAcceleration=1.396263 cartesianSpeed=0.005 cartesianAcceleration=0.01); variable=subir
                  bajada_broca := pose_sub(bajada_broca, bajada)
                MoveDirectionNode (selectedDirection=ZPlus toolParams=0.03, 0.035)
                  Until DISTANCE (allowActions=false deceleration=3 distanceNodeType=STOP) Distance=0.06; motionParameters(blendRadius=0)
                Set DigitalOutput pin=config_out[1]; digitalValue=0
                barreno_actual := barreno_actual+1
                Call Quitar_broca
                Call Poner_broca
      Popup Message (haltProgram=false message=Linea1 con full Terminada! inputType=Text)
      Folder Linea2
        Folder Marcar_puntos
          MoveL speed 100 mm/s, acceleration 500 mm/s^2 (useActiveTCP=true) feature=Base
            Waypoint punto_inicio1: TCP in base x=646.451 y=-11.704 z=260.166 mm, rx=2.1511 ry=2.2897 rz=0 rad; joints [-205.616, -96.356, 115.768, -18.693, -308.324, -0.329] deg; TCP offset x=0.411 y=-218.298 z=37.994 mm, rx=1.558 ry=-0.1255 rz=0.1212 rad
            Waypoint Linea2_A: TCP in base x=466.152 y=180.095 z=80.596 mm, rx=2.7092 ry=1.5752 rz=0.0035 rad; joints [-170.07, -97.302, 137.574, -40.225, -239.59, -0.018] deg; TCP offset x=0.411 y=-218.298 z=37.994 mm, rx=1.558 ry=-0.1255 rz=0.1212 rad
            Waypoint Linea2_B referenceName=Linea2_B: TCP in base x=669.642 y=179.866 z=80.737 mm, rx=2.7092 ry=1.5752 rz=0.0035 rad; joints [-173.706, -79.789, 119.419, -39.574, -243.231, -0.007] deg
            Waypoint Linea2_C: TCP in base x=694.939 y=178.643 z=80.843 mm, rx=2.7092 ry=1.5752 rz=0.0035 rad; joints [-174.103, -77.842, 116.933, -39.035, -243.627, -0.006] deg
            Waypoint Linea2_D: TCP in base x=897.97 y=178.427 z=80.373 mm, rx=2.7092 ry=1.5752 rz=0.0035 rad; joints [-175.658, -62.16, 94.258, -32.04, -245.171, -0.008] deg
            Waypoint Linea2_E referenceName=Linea2_E: TCP in base x=923.127 y=178.076 z=79.947 mm, rx=2.7092 ry=1.5752 rz=0.0035 rad; joints [-175.819, -60.176, 91.121, -30.888, -245.33, -0.008] deg
            Waypoint Linea2_F: TCP in base x=1151.498 y=177.179 z=80.752 mm, rx=2.7092 ry=1.5752 rz=0.0035 rad; joints [-176.803, -39.928, 55.644, -15.661, -246.279, -0.017] deg
        Folder AB
          'desbaste_inicial'
          bajada_broca := p[0,0,-0.012,0,0,0]
          barrenos_menos1 := 8
          barreno_actual := 0
          Loop While (checkContinuously=false) expression=barreno_actual≤barrenos_menos1
            Folder Perforacion
              MoveL speed 100 mm/s, acceleration 500 mm/s^2 (useActiveTCP=true) feature=Base
                internos := interpolate_pose(Linea2_A, Linea2_B, barreno_actual/barrenos_menos1)
                Waypoint Waypoint (Variable): variable=internos
                'desbaste_inicial'
                bajada_broca := p[0,0,-0.012,0,0,0]
                bajada := p[0,0,0.012,0,0,0]
                MoveDirectionNode (selectedDirection=ZMinus toolParams=0.02, 0.015)
                  Until DISTANCE (allowActions=false deceleration=3 distanceNodeType=STOP) Distance=0.055; motionParameters(blendRadius=0)
                Popup Message (haltProgram=false message=punto contacto alanzdo inputType=Text)
                MoveDirectionNode (selectedDirection=ZPlus toolParams=0.003, 0.005)
                  Until DISTANCE (allowActions=false deceleration=3 distanceNodeType=STOP) Distance=0.001; motionParameters(blendRadius=0)
                Wait Sleep waitTime=0.3
                Set DigitalOutput pin=config_out[1]; digitalValue=1
                Wait Sleep waitTime=0.3
                Loop Counting (count=2) loopVariable(name=Loop_40)
                  bajar := pose_add(get_actual_tcp_pose(), bajada_broca)
                  Waypoint Waypoint (Variable): motionParameters(jointSpeed=1.047198 jointAcceleration=1.396263 cartesianSpeed=0.001 cartesianAcceleration=0.005); variable=bajar
                  subir := pose_sub(get_actual_tcp_pose(), bajada_broca)
                  Waypoint Waypoint (Variable): motionParameters(jointSpeed=1.047198 jointAcceleration=1.396263 cartesianSpeed=0.005 cartesianAcceleration=0.01); variable=subir
                  bajada_broca := pose_sub(bajada_broca, bajada)
                MoveDirectionNode (selectedDirection=ZPlus toolParams=0.03, 0.035)
                  Until DISTANCE (allowActions=false deceleration=3 distanceNodeType=STOP) Distance=0.06; motionParameters(blendRadius=0)
                Set DigitalOutput pin=config_out[1]; digitalValue=0
                barreno_actual := barreno_actual+1
                Call Quitar_broca
                Call Poner_broca
        Folder CD
          'desbaste_inicial'
          bajada_broca := p[0,0,-0.012,0,0,0]
          barrenos_menos1 := 8
          barreno_actual := 0
          Loop While (checkContinuously=false) expression=barreno_actual≤barrenos_menos1
            Folder Perforacion
              MoveL speed 100 mm/s, acceleration 500 mm/s^2 (useActiveTCP=true) feature=Base
                internos := interpolate_pose(Linea2_C, Linea2_D, barreno_actual/barrenos_menos1)
                Waypoint Waypoint (Variable): variable=internos
                'desbaste_inicial'
                bajada_broca := p[0,0,-0.012,0,0,0]
                bajada := p[0,0,0.012,0,0,0]
                MoveDirectionNode (selectedDirection=ZMinus toolParams=0.02, 0.025)
                  Until DISTANCE (allowActions=false deceleration=3 distanceNodeType=STOP) Distance=0.055; motionParameters(blendRadius=0)
                Popup Message (haltProgram=false message=punto contacto alanzdo inputType=Text)
                MoveDirectionNode (selectedDirection=ZPlus toolParams=0.003, 0.005)
                  Until DISTANCE (allowActions=false deceleration=3 distanceNodeType=STOP) Distance=0.001; motionParameters(blendRadius=0)
                Wait Sleep waitTime=0.3
                Set DigitalOutput pin=config_out[1]; digitalValue=1
                Wait Sleep waitTime=0.3
                Loop Counting (count=2) loopVariable(name=Loop_42)
                  bajar := pose_add(get_actual_tcp_pose(), bajada_broca)
                  Waypoint Waypoint (Variable): motionParameters(jointSpeed=1.047198 jointAcceleration=1.396263 cartesianSpeed=0.001 cartesianAcceleration=0.005); variable=bajar
                  subir := pose_sub(get_actual_tcp_pose(), bajada_broca)
                  Waypoint Waypoint (Variable): motionParameters(jointSpeed=1.047198 jointAcceleration=1.396263 cartesianSpeed=0.005 cartesianAcceleration=0.01); variable=subir
                  bajada_broca := pose_sub(bajada_broca, bajada)
                MoveDirectionNode (selectedDirection=ZPlus toolParams=0.03, 0.035)
                  Until DISTANCE (allowActions=false deceleration=3 distanceNodeType=STOP) Distance=0.06; motionParameters(blendRadius=0)
                Set DigitalOutput pin=config_out[1]; digitalValue=0
                barreno_actual := barreno_actual+1
                Call Quitar_broca
                Call Poner_broca
        Folder EF
          'desbaste_inicial'
          bajada_broca := p[0,0,-0.012,0,0,0]
          barrenos_menos1 := 9
          barreno_actual := 0
          Loop While (checkContinuously=false) expression=barreno_actual≤barrenos_menos1
            Folder Perforacion
              MoveL speed 100 mm/s, acceleration 500 mm/s^2 (useActiveTCP=true) feature=Base
                internos := interpolate_pose(Linea2_E, Linea2_F, barreno_actual/barrenos_menos1)
                Waypoint Waypoint (Variable): variable=internos
                'desbaste_inicial'
                bajada_broca := p[0,0,-0.012,0,0,0]
                bajada := p[0,0,0.012,0,0,0]
                MoveDirectionNode (selectedDirection=ZMinus toolParams=0.02, 0.025)
                  Until DISTANCE (allowActions=false deceleration=3 distanceNodeType=STOP) Distance=0.055; motionParameters(blendRadius=0)
                Popup Message (haltProgram=false message=punto contacto alanzdo inputType=Text)
                MoveDirectionNode (selectedDirection=ZPlus toolParams=0.003, 0.005)
                  Until DISTANCE (allowActions=false deceleration=3 distanceNodeType=STOP) Distance=0.001; motionParameters(blendRadius=0)
                Wait Sleep waitTime=0.3
                Set DigitalOutput pin=config_out[1]; digitalValue=1
                Wait Sleep waitTime=0.3
                Loop Counting (count=2) loopVariable(name=Loop_44)
                  bajar := pose_add(get_actual_tcp_pose(), bajada_broca)
                  Waypoint Waypoint (Variable): motionParameters(jointSpeed=1.047198 jointAcceleration=1.396263 cartesianSpeed=0.001 cartesianAcceleration=0.005); variable=bajar
                  subir := pose_sub(get_actual_tcp_pose(), bajada_broca)
                  Waypoint Waypoint (Variable): motionParameters(jointSpeed=1.047198 jointAcceleration=1.396263 cartesianSpeed=0.005 cartesianAcceleration=0.01); variable=subir
                  bajada_broca := pose_sub(bajada_broca, bajada)
                MoveDirectionNode (selectedDirection=ZPlus toolParams=0.03, 0.035)
                  Until DISTANCE (allowActions=false deceleration=3 distanceNodeType=STOP) Distance=0.06; motionParameters(blendRadius=0)
                Set DigitalOutput pin=config_out[1]; digitalValue=0
                barreno_actual := barreno_actual+1
                If barreno_actual>barrenos_menos1
                  cambiar_broca := True
                Call Quitar_broca
                Call Poner_broca
      Popup Message (haltProgram=false message=Linea2 con full Terminada! inputType=Text)
  Folder Posicion3
    eje7 := 3
    Folder Broca_1
      Folder Linea3
        Folder Marcar_puntos
          MoveL speed 100 mm/s, acceleration 500 mm/s^2 (useActiveTCP=true) feature=Base
            Waypoint punto_inicio1: TCP in base x=646.451 y=-11.704 z=260.166 mm, rx=2.1511 ry=2.2897 rz=0 rad; joints [-205.616, -96.356, 115.768, -18.693, -308.324, -0.329] deg; TCP offset x=0.411 y=-218.298 z=37.994 mm, rx=1.558 ry=-0.1255 rz=0.1212 rad
            Waypoint Linea3_A: TCP in base x=460.55 y=-395.563 z=80.682 mm, rx=3.1326 ry=-0.0943 rz=0.0057 rad; joints [-228.865, -86.051, 126.783, -40.72, -234.593, 0.309] deg; TCP offset x=0.411 y=-218.298 z=37.994 mm, rx=1.558 ry=-0.1255 rz=0.1212 rad
            Waypoint Linea3_B: TCP in base x=664.301 y=-395.445 z=81.308 mm, rx=3.1326 ry=-0.0943 rz=0.0057 rad; joints [-215.162, -70.126, 106.29, -36.16, -220.885, 0.318] deg
            Waypoint Linea3_C: TCP in base x=689.223 y=-395.791 z=80.699 mm, rx=3.1326 ry=-0.0943 rz=0.0057 rad; joints [-213.996, -68.184, 103.511, -35.323, -219.718, 0.318] deg
            Waypoint Linea3_D: TCP in base x=892.727 y=-396.221 z=80.325 mm, rx=3.1326 ry=-0.0943 rz=0.0057 rad; joints [-206.597, -52.057, 77.467, -25.419, -212.299, 0.312] deg
            Waypoint Linea3_E: TCP in base x=918.375 y=-396.594 z=80.115 mm, rx=3.1326 ry=-0.0943 rz=0.0057 rad; joints [-205.9, -49.825, 73.601, -23.787, -211.599, 0.31] deg
            Waypoint Linea3_F: TCP in base x=1146.287 y=-396.633 z=80.258 mm, rx=3.1324 ry=-0.0938 rz=0.0063 rad; joints [-200.88, -21.042, 19.258, 1.725, -206.53, 0.288] deg; TCP offset x=0.411 y=-218.298 z=37.994 mm, rx=1.558 ry=-0.1255 rz=0.1212 rad
        Folder AB
          'desbaste_inicial'
          bajada_broca := p[0,0,-0.008,0,0,0]
          barrenos_menos1 := 8
          barreno_actual := 0
          Loop While (checkContinuously=false) expression=barreno_actual≤barrenos_menos1
            Folder Perforacion
              MoveL speed 100 mm/s, acceleration 500 mm/s^2 (useActiveTCP=true) feature=Base
                internos := interpolate_pose(Linea3_A, Linea3_B, barreno_actual/barrenos_menos1)
                Waypoint Waypoint (Variable): variable=internos
                'desbaste_inicial'
                bajada_broca := p[0,0,-0.008,0,0,0]
                bajada := p[0,0,0.008,0,0,0]
                MoveDirectionNode (selectedDirection=ZMinus toolParams=0.02, 0.015)
                  Until DISTANCE (allowActions=false deceleration=3 distanceNodeType=STOP) Distance=0.055; motionParameters(blendRadius=0)
                Popup Message (haltProgram=false message=punto contacto alanzdo inputType=Text)
                MoveDirectionNode (selectedDirection=ZPlus toolParams=0.003, 0.005)
                  Until DISTANCE (allowActions=false deceleration=3 distanceNodeType=STOP) Distance=0.001; motionParameters(blendRadius=0)
                Wait Sleep waitTime=0.3
                Set DigitalOutput pin=config_out[1]; digitalValue=1
                Wait Sleep waitTime=0.3
                Loop Counting (count=3) loopVariable(name=Loop_26)
                  bajar := pose_add(get_actual_tcp_pose(), bajada_broca)
                  Waypoint Waypoint (Variable): motionParameters(jointSpeed=1.047198 jointAcceleration=1.396263 cartesianSpeed=0.001 cartesianAcceleration=0.005); variable=bajar
                  subir := pose_sub(get_actual_tcp_pose(), bajada_broca)
                  Waypoint Waypoint (Variable): motionParameters(jointSpeed=1.047198 jointAcceleration=1.396263 cartesianSpeed=0.005 cartesianAcceleration=0.01); variable=subir
                  bajada_broca := pose_sub(bajada_broca, bajada)
                MoveDirectionNode (selectedDirection=ZPlus toolParams=0.03, 0.035)
                  Until DISTANCE (allowActions=false deceleration=3 distanceNodeType=STOP) Distance=0.06; motionParameters(blendRadius=0)
                Set DigitalOutput pin=config_out[1]; digitalValue=0
                barreno_actual := barreno_actual+1
                Call Quitar_broca
                Call Poner_broca
        Folder CD
          'desbaste_inicial'
          bajada_broca := p[0,0,-0.008,0,0,0]
          barrenos_menos1 := 8
          barreno_actual := 0
          Loop While (checkContinuously=false) expression=barreno_actual≤barrenos_menos1
            Folder Perforacion
              MoveL speed 100 mm/s, acceleration 500 mm/s^2 (useActiveTCP=true) feature=Base
                internos := interpolate_pose(Linea3_C, Linea3_D, barreno_actual/barrenos_menos1)
                Waypoint Waypoint (Variable): variable=internos
                'desbaste_inicial'
                bajada_broca := p[0,0,-0.008,0,0,0]
                bajada := p[0,0,0.008,0,0,0]
                MoveDirectionNode (selectedDirection=ZMinus toolParams=0.015, 0.02)
                  Until DISTANCE (allowActions=false deceleration=3 distanceNodeType=STOP) Distance=0.055; motionParameters(blendRadius=0)
                Popup Message (haltProgram=false message=punto contacto alanzdo inputType=Text)
                MoveDirectionNode (selectedDirection=ZPlus toolParams=0.003, 0.005)
                  Until DISTANCE (allowActions=false deceleration=3 distanceNodeType=STOP) Distance=0.001; motionParameters(blendRadius=0)
                Wait Sleep waitTime=0.3
                Set DigitalOutput pin=config_out[1]; digitalValue=1
                Wait Sleep waitTime=0.3
                Loop Counting (count=3) loopVariable(name=Loop_28)
                  bajar := pose_add(get_actual_tcp_pose(), bajada_broca)
                  Waypoint Waypoint (Variable): motionParameters(jointSpeed=1.047198 jointAcceleration=1.396263 cartesianSpeed=0.001 cartesianAcceleration=0.005); variable=bajar
                  subir := pose_sub(get_actual_tcp_pose(), bajada_broca)
                  Waypoint Waypoint (Variable): motionParameters(jointSpeed=1.047198 jointAcceleration=1.396263 cartesianSpeed=0.005 cartesianAcceleration=0.01); variable=subir
                  bajada_broca := pose_sub(bajada_broca, bajada)
                MoveDirectionNode (selectedDirection=ZPlus toolParams=0.03, 0.035)
                  Until DISTANCE (allowActions=false deceleration=3 distanceNodeType=STOP) Distance=0.06; motionParameters(blendRadius=0)
                Set DigitalOutput pin=config_out[1]; digitalValue=0
                barreno_actual := barreno_actual+1
                Call Quitar_broca
                Call Poner_broca
        Folder EF
          'desbaste_inicial'
          bajada_broca := p[0,0,-0.008,0,0,0]
          barrenos_menos1 := 9
          barreno_actual := 0
          Loop While (checkContinuously=false) expression=barreno_actual≤barrenos_menos1
            Folder Perforacion
              MoveL speed 100 mm/s, acceleration 500 mm/s^2 (useActiveTCP=true) feature=Base
                internos := interpolate_pose(Linea3_E, Linea3_F, barreno_actual/barrenos_menos1)
                Waypoint Waypoint (Variable): variable=internos
                'desbaste_inicial'
                bajada_broca := p[0,0,-0.008,0,0,0]
                bajada := p[0,0,0.008,0,0,0]
                MoveDirectionNode (selectedDirection=ZMinus toolParams=0.02, 0.015)
                  Until DISTANCE (allowActions=false deceleration=3 distanceNodeType=STOP) Distance=0.055; motionParameters(blendRadius=0)
                Popup Message (haltProgram=false message=punto contacto alanzdo inputType=Text)
                MoveDirectionNode (selectedDirection=ZPlus toolParams=0.003, 0.005)
                  Until DISTANCE (allowActions=false deceleration=3 distanceNodeType=STOP) Distance=0.001; motionParameters(blendRadius=0)
                Wait Sleep waitTime=0.3
                Set DigitalOutput pin=config_out[1]; digitalValue=1
                Wait Sleep waitTime=0.3
                Loop Counting (count=3) loopVariable(name=Loop_30)
                  bajar := pose_add(get_actual_tcp_pose(), bajada_broca)
                  Waypoint Waypoint (Variable): motionParameters(jointSpeed=1.047198 jointAcceleration=1.396263 cartesianSpeed=0.001 cartesianAcceleration=0.005); variable=bajar
                  subir := pose_sub(get_actual_tcp_pose(), bajada_broca)
                  Waypoint Waypoint (Variable): motionParameters(jointSpeed=1.047198 jointAcceleration=1.396263 cartesianSpeed=0.005 cartesianAcceleration=0.01); variable=subir
                  bajada_broca := pose_sub(bajada_broca, bajada)
                MoveDirectionNode (selectedDirection=ZPlus toolParams=0.03, 0.035)
                  Until DISTANCE (allowActions=false deceleration=3 distanceNodeType=STOP) Distance=0.06; motionParameters(blendRadius=0)
                Set DigitalOutput pin=config_out[1]; digitalValue=0
                barreno_actual := barreno_actual+1
                Call Quitar_broca
                Call Poner_broca
      Popup Message (haltProgram=false message=Linea1 con chica Terminada! inputType=Text)
      Folder Linea4
        Folder Marcar_puntos
          MoveL speed 100 mm/s, acceleration 500 mm/s^2 (useActiveTCP=true) feature=Base
            Waypoint punto_inicio1: TCP in base x=646.451 y=-11.704 z=260.166 mm, rx=2.1511 ry=2.2897 rz=0 rad; joints [-205.616, -96.356, 115.768, -18.693, -308.324, -0.329] deg; TCP offset x=0.411 y=-218.298 z=37.994 mm, rx=1.558 ry=-0.1255 rz=0.1212 rad
            Waypoint Linea4_A: TCP in base x=464.055 y=12.985 z=80.074 mm, rx=2.5347 ry=1.8484 rz=0.0134 rad; joints [-207.418, -108.682, 145.56, -36.88, -288.784, 0.283] deg; TCP offset x=0.411 y=-218.298 z=37.994 mm, rx=1.558 ry=-0.1255 rz=0.1212 rad
            Waypoint Linea4_B: TCP in base x=667.246 y=12.985 z=80.29 mm, rx=2.5347 ry=1.8484 rz=0.0134 rad; joints [-195.874, -85.057, 125.756, -40.72, -277.256, 0.307] deg
            Waypoint Linea4_C: TCP in base x=692.679 y=13.033 z=80.385 mm, rx=2.5347 ry=1.8484 rz=0.0134 rad; joints [-195.088, -82.745, 123.085, -40.362, -276.469, 0.308] deg
            Waypoint Linea4_D: TCP in base x=895.963 y=12.684 z=81.163 mm, rx=2.5347 ry=1.8484 rz=0.0134 rad; joints [-190.876, -65.82, 99.909, -34.115, -272.249, 0.309] deg
            Waypoint Linea4_E: TCP in base x=921.05 y=12.352 z=81.665 mm, rx=2.5347 ry=1.8484 rz=0.0134 rad; joints [-190.538, -63.815, 96.748, -32.958, -271.909, 0.308] deg
            Waypoint Linea4_F: TCP in base x=1149.402 y=11.805 z=82.23 mm, rx=2.5347 ry=1.8484 rz=0.0134 rad; joints [-188.123, -43.805, 62.636, -18.859, -269.462, 0.301] deg
        Folder AB
          'desbaste_inicial'
          bajada_broca := p[0,0,-0.008,0,0,0]
          barrenos_menos1 := 8
          barreno_actual := 0
          Loop While (checkContinuously=false) expression=barreno_actual≤barrenos_menos1
            Folder Perforacion
              MoveL speed 100 mm/s, acceleration 500 mm/s^2 (useActiveTCP=true) feature=Base
                internos := interpolate_pose(Linea4_A, Linea4_B, barreno_actual/barrenos_menos1)
                Waypoint Waypoint (Variable): variable=internos
                'desbaste_inicial'
                bajada_broca := p[0,0,-0.008,0,0,0]
                bajada := p[0,0,0.008,0,0,0]
                MoveDirectionNode (selectedDirection=ZMinus toolParams=0.02, 0.015)
                  Until DISTANCE (allowActions=false deceleration=3 distanceNodeType=STOP) Distance=0.055; motionParameters(blendRadius=0)
                Popup Message (haltProgram=false message=punto contacto alanzdo inputType=Text)
                MoveDirectionNode (selectedDirection=ZPlus toolParams=0.003, 0.005)
                  Until DISTANCE (allowActions=false deceleration=3 distanceNodeType=STOP) Distance=0.002; motionParameters(blendRadius=0)
                Wait Sleep waitTime=0.3
                Set DigitalOutput pin=config_out[1]; digitalValue=1
                Wait Sleep waitTime=0.3
                Loop Counting (count=3) loopVariable(name=Loop_32)
                  bajar := pose_add(get_actual_tcp_pose(), bajada_broca)
                  Waypoint Waypoint (Variable): motionParameters(jointSpeed=1.047198 jointAcceleration=1.396263 cartesianSpeed=0.001 cartesianAcceleration=0.005); variable=bajar
                  subir := pose_sub(get_actual_tcp_pose(), bajada_broca)
                  Waypoint Waypoint (Variable): motionParameters(jointSpeed=1.047198 jointAcceleration=1.396263 cartesianSpeed=0.005 cartesianAcceleration=0.01); variable=subir
                  bajada_broca := pose_sub(bajada_broca, bajada)
                MoveDirectionNode (selectedDirection=ZPlus toolParams=0.03, 0.035)
                  Until DISTANCE (allowActions=false deceleration=3 distanceNodeType=STOP) Distance=0.06; motionParameters(blendRadius=0)
                Set DigitalOutput pin=config_out[1]; digitalValue=0
                barreno_actual := barreno_actual+1
                SuppressedNode
                  Call Quitar_broca
                SuppressedNode
                  Call Poner_broca
        Folder CD
          'desbaste_inicial'
          bajada_broca := p[0,0,-0.008,0,0,0]
          barrenos_menos1 := 8
          barreno_actual := 0
          Loop While (checkContinuously=false) expression=barreno_actual≤barrenos_menos1
            Folder Perforacion
              MoveL speed 100 mm/s, acceleration 500 mm/s^2 (useActiveTCP=true) feature=Base
                internos := interpolate_pose(Linea4_C, Linea4_D, barreno_actual/barrenos_menos1)
                Waypoint Waypoint (Variable): variable=internos
                'desbaste_inicial'
                bajada_broca := p[0,0,-0.008,0,0,0]
                bajada := p[0,0,0.008,0,0,0]
                MoveDirectionNode (selectedDirection=ZMinus toolParams=0.02, 0.015)
                  Until DISTANCE (allowActions=false deceleration=3 distanceNodeType=STOP) Distance=0.055; motionParameters(blendRadius=0)
                Popup Message (haltProgram=false message=punto contacto alanzdo inputType=Text)
                MoveDirectionNode (selectedDirection=ZPlus toolParams=0.003, 0.005)
                  Until DISTANCE (allowActions=false deceleration=3 distanceNodeType=STOP) Distance=0.002; motionParameters(blendRadius=0)
                Wait Sleep waitTime=0.3
                Set DigitalOutput pin=config_out[1]; digitalValue=1
                Wait Sleep waitTime=0.3
                Loop Counting (count=3) loopVariable(name=Loop_35)
                  bajar := pose_add(get_actual_tcp_pose(), bajada_broca)
                  Waypoint Waypoint (Variable): motionParameters(jointSpeed=1.047198 jointAcceleration=1.396263 cartesianSpeed=0.001 cartesianAcceleration=0.005); variable=bajar
                  subir := pose_sub(get_actual_tcp_pose(), bajada_broca)
                  Waypoint Waypoint (Variable): motionParameters(jointSpeed=1.047198 jointAcceleration=1.396263 cartesianSpeed=0.005 cartesianAcceleration=0.01); variable=subir
                  bajada_broca := pose_sub(bajada_broca, bajada)
                MoveDirectionNode (selectedDirection=ZPlus toolParams=0.03, 0.035)
                  Until DISTANCE (allowActions=false deceleration=3 distanceNodeType=STOP) Distance=0.06; motionParameters(blendRadius=0)
                Set DigitalOutput pin=config_out[1]; digitalValue=0
                barreno_actual := barreno_actual+1
                SuppressedNode
                  Call Quitar_broca
                SuppressedNode
                  Call Poner_broca
        Folder EF
          'desbaste_inicial'
          bajada_broca := p[0,0,-0.008,0,0,0]
          barrenos_menos1 := 9
          barreno_actual := 0
          Loop While (checkContinuously=false) expression=barreno_actual≤barrenos_menos1
            Folder Perforacion
              MoveL speed 100 mm/s, acceleration 500 mm/s^2 (useActiveTCP=true) feature=Base
                internos := interpolate_pose(Linea4_E, Linea4_F, barreno_actual/barrenos_menos1)
                Waypoint Waypoint (Variable): variable=internos
                'desbaste_inicial'
                bajada_broca := p[0,0,-0.008,0,0,0]
                bajada := p[0,0,0.008,0,0,0]
                MoveDirectionNode (selectedDirection=ZMinus toolParams=0.02, 0.015)
                  Until DISTANCE (allowActions=false deceleration=3 distanceNodeType=STOP) Distance=0.055; motionParameters(blendRadius=0)
                Popup Message (haltProgram=false message=punto contacto alanzdo inputType=Text)
                MoveDirectionNode (selectedDirection=ZPlus toolParams=0.003, 0.005)
                  Until DISTANCE (allowActions=false deceleration=3 distanceNodeType=STOP) Distance=0.002; motionParameters(blendRadius=0)
                Wait Sleep waitTime=0.3
                Set DigitalOutput pin=config_out[1]; digitalValue=1
                Wait Sleep waitTime=0.3
                Loop Counting (count=3) loopVariable(name=Loop_39)
                  bajar := pose_add(get_actual_tcp_pose(), bajada_broca)
                  Waypoint Waypoint (Variable): motionParameters(jointSpeed=1.047198 jointAcceleration=1.396263 cartesianSpeed=0.001 cartesianAcceleration=0.005); variable=bajar
                  subir := pose_sub(get_actual_tcp_pose(), bajada_broca)
                  Waypoint Waypoint (Variable): motionParameters(jointSpeed=1.047198 jointAcceleration=1.396263 cartesianSpeed=0.005 cartesianAcceleration=0.01); variable=subir
                  bajada_broca := pose_sub(bajada_broca, bajada)
                MoveDirectionNode (selectedDirection=ZPlus toolParams=0.03, 0.035)
                  Until DISTANCE (allowActions=false deceleration=3 distanceNodeType=STOP) Distance=0.06; motionParameters(blendRadius=0)
                Set DigitalOutput pin=config_out[1]; digitalValue=0
                barreno_actual := barreno_actual+1
                If barreno_actual>barrenos_menos1
                  cambiar_broca := True
                SuppressedNode
                  Call Quitar_broca
                SuppressedNode
                  Call Poner_broca
      Popup Message (haltProgram=false message=Linea2 con chica Terminada! inputType=Text)
    Folder Broca_2
      Folder Linea3
        Folder Marcar_puntos
          MoveL speed 100 mm/s, acceleration 500 mm/s^2 (useActiveTCP=true) feature=Base
            Waypoint punto_inicio1: TCP in base x=646.451 y=-11.704 z=260.166 mm, rx=2.1511 ry=2.2897 rz=0 rad; joints [-205.616, -96.356, 115.768, -18.693, -308.324, -0.329] deg; TCP offset x=0.411 y=-218.298 z=37.994 mm, rx=1.558 ry=-0.1255 rz=0.1212 rad
            Waypoint Linea3_A: TCP in base x=460.55 y=-395.563 z=80.682 mm, rx=3.1326 ry=-0.0943 rz=0.0057 rad; joints [-228.865, -86.051, 126.783, -40.72, -234.593, 0.309] deg; TCP offset x=0.411 y=-218.298 z=37.994 mm, rx=1.558 ry=-0.1255 rz=0.1212 rad
            Waypoint Linea3_B: TCP in base x=664.301 y=-395.445 z=81.308 mm, rx=3.1326 ry=-0.0943 rz=0.0057 rad; joints [-215.162, -70.126, 106.29, -36.16, -220.885, 0.318] deg
            Waypoint Linea3_C: TCP in base x=689.223 y=-395.791 z=80.699 mm, rx=3.1326 ry=-0.0943 rz=0.0057 rad; joints [-213.996, -68.184, 103.511, -35.323, -219.718, 0.318] deg
            Waypoint Linea3_D: TCP in base x=892.727 y=-396.221 z=80.325 mm, rx=3.1326 ry=-0.0943 rz=0.0057 rad; joints [-206.597, -52.057, 77.467, -25.419, -212.299, 0.312] deg
            Waypoint Linea3_E: TCP in base x=918.375 y=-396.594 z=80.115 mm, rx=3.1326 ry=-0.0943 rz=0.0057 rad; joints [-205.9, -49.825, 73.601, -23.787, -211.599, 0.31] deg
            Waypoint Linea3_F: TCP in base x=1146.287 y=-396.633 z=80.258 mm, rx=3.1324 ry=-0.0938 rz=0.0063 rad; joints [-200.88, -21.042, 19.258, 1.725, -206.53, 0.288] deg; TCP offset x=0.411 y=-218.298 z=37.994 mm, rx=1.558 ry=-0.1255 rz=0.1212 rad
        Folder AB
          'desbaste_inicial'
          bajada_broca := p[0,0,-0.012,0,0,0]
          barrenos_menos1 := 8
          barreno_actual := 0
          Loop While (checkContinuously=false) expression=barreno_actual≤barrenos_menos1
            Folder Perforacion
              MoveL speed 100 mm/s, acceleration 500 mm/s^2 (useActiveTCP=true) feature=Base
                internos := interpolate_pose(Linea3_A, Linea3_B, barreno_actual/barrenos_menos1)
                Waypoint Waypoint (Variable): variable=internos
                'desbaste_inicial'
                bajada_broca := p[0,0,-0.012,0,0,0]
                bajada := p[0,0,0.012,0,0,0]
                MoveDirectionNode (selectedDirection=ZMinus toolParams=0.02, 0.015)
                  Until DISTANCE (allowActions=false deceleration=3 distanceNodeType=STOP) Distance=0.055; motionParameters(blendRadius=0)
                Popup Message (haltProgram=false message=punto contacto alanzdo inputType=Text)
                MoveDirectionNode (selectedDirection=ZPlus toolParams=0.003, 0.005)
                  Until DISTANCE (allowActions=false deceleration=3 distanceNodeType=STOP) Distance=0.002; motionParameters(blendRadius=0)
                Wait Sleep waitTime=0.3
                Set DigitalOutput pin=config_out[1]; digitalValue=1
                Wait Sleep waitTime=0.3
                Loop Counting (count=2) loopVariable(name=Loop_70)
                  bajar := pose_add(get_actual_tcp_pose(), bajada_broca)
                  Waypoint Waypoint (Variable): motionParameters(jointSpeed=1.047198 jointAcceleration=1.396263 cartesianSpeed=0.001 cartesianAcceleration=0.005); variable=bajar
                  subir := pose_sub(get_actual_tcp_pose(), bajada_broca)
                  Waypoint Waypoint (Variable): motionParameters(jointSpeed=1.047198 jointAcceleration=1.396263 cartesianSpeed=0.005 cartesianAcceleration=0.01); variable=subir
                  bajada_broca := pose_sub(bajada_broca, bajada)
                MoveDirectionNode (selectedDirection=ZPlus toolParams=0.03, 0.035)
                  Until DISTANCE (allowActions=false deceleration=3 distanceNodeType=STOP) Distance=0.06; motionParameters(blendRadius=0)
                Set DigitalOutput pin=config_out[1]; digitalValue=0
                barreno_actual := barreno_actual+1
                SuppressedNode
                  Call Quitar_broca
                SuppressedNode
                  Call Poner_broca
        Folder CD
          'desbaste_inicial'
          bajada_broca := p[0,0,-0.012,0,0,0]
          barrenos_menos1 := 8
          barreno_actual := 0
          Loop While (checkContinuously=false) expression=barreno_actual≤barrenos_menos1
            Folder Perforacion
              MoveL speed 100 mm/s, acceleration 500 mm/s^2 (useActiveTCP=true) feature=Base
                internos := interpolate_pose(Linea3_C, Linea3_D, barreno_actual/barrenos_menos1)
                Waypoint Waypoint (Variable): variable=internos
                'desbaste_inicial'
                bajada_broca := p[0,0,-0.012,0,0,0]
                bajada := p[0,0,0.012,0,0,0]
                MoveDirectionNode (selectedDirection=ZMinus toolParams=0.015, 0.02)
                  Until DISTANCE (allowActions=false deceleration=3 distanceNodeType=STOP) Distance=0.055; motionParameters(blendRadius=0)
                Popup Message (haltProgram=false message=punto contacto alanzdo inputType=Text)
                MoveDirectionNode (selectedDirection=ZPlus toolParams=0.003, 0.005)
                  Until DISTANCE (allowActions=false deceleration=3 distanceNodeType=STOP) Distance=0.002; motionParameters(blendRadius=0)
                Wait Sleep waitTime=0.3
                Set DigitalOutput pin=config_out[1]; digitalValue=1
                Wait Sleep waitTime=0.3
                Loop Counting (count=2) loopVariable(name=Loop_72)
                  bajar := pose_add(get_actual_tcp_pose(), bajada_broca)
                  Waypoint Waypoint (Variable): motionParameters(jointSpeed=1.047198 jointAcceleration=1.396263 cartesianSpeed=0.001 cartesianAcceleration=0.005); variable=bajar
                  subir := pose_sub(get_actual_tcp_pose(), bajada_broca)
                  Waypoint Waypoint (Variable): motionParameters(jointSpeed=1.047198 jointAcceleration=1.396263 cartesianSpeed=0.005 cartesianAcceleration=0.01); variable=subir
                  bajada_broca := pose_sub(bajada_broca, bajada)
                MoveDirectionNode (selectedDirection=ZPlus toolParams=0.03, 0.035)
                  Until DISTANCE (allowActions=false deceleration=3 distanceNodeType=STOP) Distance=0.06; motionParameters(blendRadius=0)
                Set DigitalOutput pin=config_out[1]; digitalValue=0
                barreno_actual := barreno_actual+1
                SuppressedNode
                  Call Quitar_broca
                SuppressedNode
                  Call Poner_broca
        Folder EF
          'desbaste_inicial'
          bajada_broca := p[0,0,-0.012,0,0,0]
          barrenos_menos1 := 9
          barreno_actual := 0
          Loop While (checkContinuously=false) expression=barreno_actual≤barrenos_menos1
            Folder Perforacion
              MoveL speed 100 mm/s, acceleration 500 mm/s^2 (useActiveTCP=true) feature=Base
                internos := interpolate_pose(Linea3_E, Linea3_F, barreno_actual/barrenos_menos1)
                Waypoint Waypoint (Variable): variable=internos
                'desbaste_inicial'
                bajada_broca := p[0,0,-0.012,0,0,0]
                bajada := p[0,0,0.012,0,0,0]
                MoveDirectionNode (selectedDirection=ZMinus toolParams=0.02, 0.015)
                  Until DISTANCE (allowActions=false deceleration=3 distanceNodeType=STOP) Distance=0.055; motionParameters(blendRadius=0)
                Popup Message (haltProgram=false message=punto contacto alanzdo inputType=Text)
                MoveDirectionNode (selectedDirection=ZPlus toolParams=0.003, 0.005)
                  Until DISTANCE (allowActions=false deceleration=3 distanceNodeType=STOP) Distance=0.002; motionParameters(blendRadius=0)
                Wait Sleep waitTime=0.3
                Set DigitalOutput pin=config_out[1]; digitalValue=1
                Wait Sleep waitTime=0.3
                Loop Counting (count=2) loopVariable(name=Loop_74)
                  bajar := pose_add(get_actual_tcp_pose(), bajada_broca)
                  Waypoint Waypoint (Variable): motionParameters(jointSpeed=1.047198 jointAcceleration=1.396263 cartesianSpeed=0.001 cartesianAcceleration=0.005); variable=bajar
                  subir := pose_sub(get_actual_tcp_pose(), bajada_broca)
                  Waypoint Waypoint (Variable): motionParameters(jointSpeed=1.047198 jointAcceleration=1.396263 cartesianSpeed=0.005 cartesianAcceleration=0.01); variable=subir
                  bajada_broca := pose_sub(bajada_broca, bajada)
                MoveDirectionNode (selectedDirection=ZPlus toolParams=0.03, 0.035)
                  Until DISTANCE (allowActions=false deceleration=3 distanceNodeType=STOP) Distance=0.06; motionParameters(blendRadius=0)
                Set DigitalOutput pin=config_out[1]; digitalValue=0
                barreno_actual := barreno_actual+1
                SuppressedNode
                  Call Quitar_broca
                SuppressedNode
                  Call Poner_broca
      Popup Message (haltProgram=false message=Linea1 con chica Terminada! inputType=Text)
      Folder Linea4
        Folder Marcar_puntos
          MoveL speed 100 mm/s, acceleration 500 mm/s^2 (useActiveTCP=true) feature=Base
            Waypoint punto_inicio1: TCP in base x=646.451 y=-11.704 z=260.166 mm, rx=2.1511 ry=2.2897 rz=0 rad; joints [-205.616, -96.356, 115.768, -18.693, -308.324, -0.329] deg; TCP offset x=0.411 y=-218.298 z=37.994 mm, rx=1.558 ry=-0.1255 rz=0.1212 rad
            Waypoint Linea4_A: TCP in base x=464.055 y=12.985 z=80.074 mm, rx=2.5347 ry=1.8484 rz=0.0134 rad; joints [-207.418, -108.682, 145.56, -36.88, -288.784, 0.283] deg; TCP offset x=0.411 y=-218.298 z=37.994 mm, rx=1.558 ry=-0.1255 rz=0.1212 rad
            Waypoint Linea4_B: TCP in base x=667.246 y=12.985 z=80.29 mm, rx=2.5347 ry=1.8484 rz=0.0134 rad; joints [-195.874, -85.057, 125.756, -40.72, -277.256, 0.307] deg
            Waypoint Linea4_C: TCP in base x=692.679 y=13.033 z=80.385 mm, rx=2.5347 ry=1.8484 rz=0.0134 rad; joints [-195.088, -82.745, 123.085, -40.362, -276.469, 0.308] deg
            Waypoint Linea4_D: TCP in base x=895.963 y=12.684 z=81.163 mm, rx=2.5347 ry=1.8484 rz=0.0134 rad; joints [-190.876, -65.82, 99.909, -34.115, -272.249, 0.309] deg
            Waypoint Linea4_E: TCP in base x=921.05 y=12.352 z=81.665 mm, rx=2.5347 ry=1.8484 rz=0.0134 rad; joints [-190.538, -63.815, 96.748, -32.958, -271.909, 0.308] deg
            Waypoint Linea4_F: TCP in base x=1149.402 y=11.805 z=82.23 mm, rx=2.5347 ry=1.8484 rz=0.0134 rad; joints [-188.123, -43.805, 62.636, -18.859, -269.462, 0.301] deg
        Folder AB
          'desbaste_inicial'
          bajada_broca := p[0,0,-0.012,0,0,0]
          barrenos_menos1 := 8
          barreno_actual := 0
          Loop While (checkContinuously=false) expression=barreno_actual≤barrenos_menos1
            Folder Perforacion
              MoveL speed 100 mm/s, acceleration 500 mm/s^2 (useActiveTCP=true) feature=Base
                internos := interpolate_pose(Linea4_A, Linea4_B, barreno_actual/barrenos_menos1)
                Waypoint Waypoint (Variable): variable=internos
                'desbaste_inicial'
                bajada_broca := p[0,0,-0.012,0,0,0]
                bajada := p[0,0,0.012,0,0,0]
                MoveDirectionNode (selectedDirection=ZMinus toolParams=0.02, 0.015)
                  Until DISTANCE (allowActions=false deceleration=3 distanceNodeType=STOP) Distance=0.055; motionParameters(blendRadius=0)
                Popup Message (haltProgram=false message=punto contacto alanzdo inputType=Text)
                MoveDirectionNode (selectedDirection=ZPlus toolParams=0.003, 0.005)
                  Until DISTANCE (allowActions=false deceleration=3 distanceNodeType=STOP) Distance=0.002; motionParameters(blendRadius=0)
                Wait Sleep waitTime=0.3
                Set DigitalOutput pin=config_out[1]; digitalValue=1
                Wait Sleep waitTime=0.3
                Loop Counting (count=2) loopVariable(name=Loop_76)
                  bajar := pose_add(get_actual_tcp_pose(), bajada_broca)
                  Waypoint Waypoint (Variable): motionParameters(jointSpeed=1.047198 jointAcceleration=1.396263 cartesianSpeed=0.001 cartesianAcceleration=0.005); variable=bajar
                  subir := pose_sub(get_actual_tcp_pose(), bajada_broca)
                  Waypoint Waypoint (Variable): motionParameters(jointSpeed=1.047198 jointAcceleration=1.396263 cartesianSpeed=0.005 cartesianAcceleration=0.01); variable=subir
                  bajada_broca := pose_sub(bajada_broca, bajada)
                MoveDirectionNode (selectedDirection=ZPlus toolParams=0.03, 0.035)
                  Until DISTANCE (allowActions=false deceleration=3 distanceNodeType=STOP) Distance=0.06; motionParameters(blendRadius=0)
                Set DigitalOutput pin=config_out[1]; digitalValue=0
                barreno_actual := barreno_actual+1
                SuppressedNode
                  Call Quitar_broca
                SuppressedNode
                  Call Poner_broca
        Folder CD
          'desbaste_inicial'
          bajada_broca := p[0,0,-0.012,0,0,0]
          barrenos_menos1 := 8
          barreno_actual := 0
          Loop While (checkContinuously=false) expression=barreno_actual≤barrenos_menos1
            Folder Perforacion
              MoveL speed 100 mm/s, acceleration 500 mm/s^2 (useActiveTCP=true) feature=Base
                internos := interpolate_pose(Linea4_C, Linea4_D, barreno_actual/barrenos_menos1)
                Waypoint Waypoint (Variable): variable=internos
                'desbaste_inicial'
                bajada_broca := p[0,0,-0.012,0,0,0]
                bajada := p[0,0,0.012,0,0,0]
                MoveDirectionNode (selectedDirection=ZMinus toolParams=0.02, 0.015)
                  Until DISTANCE (allowActions=false deceleration=3 distanceNodeType=STOP) Distance=0.055; motionParameters(blendRadius=0)
                Popup Message (haltProgram=false message=punto contacto alanzdo inputType=Text)
                MoveDirectionNode (selectedDirection=ZPlus toolParams=0.003, 0.005)
                  Until DISTANCE (allowActions=false deceleration=3 distanceNodeType=STOP) Distance=0.002; motionParameters(blendRadius=0)
                Wait Sleep waitTime=0.3
                Set DigitalOutput pin=config_out[1]; digitalValue=1
                Wait Sleep waitTime=0.3
                Loop Counting (count=2) loopVariable(name=Loop_78)
                  bajar := pose_add(get_actual_tcp_pose(), bajada_broca)
                  Waypoint Waypoint (Variable): motionParameters(jointSpeed=1.047198 jointAcceleration=1.396263 cartesianSpeed=0.001 cartesianAcceleration=0.005); variable=bajar
                  subir := pose_sub(get_actual_tcp_pose(), bajada_broca)
                  Waypoint Waypoint (Variable): motionParameters(jointSpeed=1.047198 jointAcceleration=1.396263 cartesianSpeed=0.005 cartesianAcceleration=0.01); variable=subir
                  bajada_broca := pose_sub(bajada_broca, bajada)
                MoveDirectionNode (selectedDirection=ZPlus toolParams=0.03, 0.035)
                  Until DISTANCE (allowActions=false deceleration=3 distanceNodeType=STOP) Distance=0.06; motionParameters(blendRadius=0)
                Set DigitalOutput pin=config_out[1]; digitalValue=0
                barreno_actual := barreno_actual+1
                SuppressedNode
                  Call Quitar_broca
                SuppressedNode
                  Call Poner_broca
        Folder EF
          'desbaste_inicial'
          bajada_broca := p[0,0,-0.012,0,0,0]
          barrenos_menos1 := 9
          barreno_actual := 0
          Loop While (checkContinuously=false) expression=barreno_actual≤barrenos_menos1
            Folder Perforacion
              MoveL speed 100 mm/s, acceleration 500 mm/s^2 (useActiveTCP=true) feature=Base
                internos := interpolate_pose(Linea4_E, Linea4_F, barreno_actual/barrenos_menos1)
                Waypoint Waypoint (Variable): variable=internos
                'desbaste_inicial'
                bajada_broca := p[0,0,-0.012,0,0,0]
                bajada := p[0,0,0.012,0,0,0]
                MoveDirectionNode (selectedDirection=ZMinus toolParams=0.02, 0.015)
                  Until DISTANCE (allowActions=false deceleration=3 distanceNodeType=STOP) Distance=0.055; motionParameters(blendRadius=0)
                Popup Message (haltProgram=false message=punto contacto alanzdo inputType=Text)
                MoveDirectionNode (selectedDirection=ZPlus toolParams=0.003, 0.005)
                  Until DISTANCE (allowActions=false deceleration=3 distanceNodeType=STOP) Distance=0.002; motionParameters(blendRadius=0)
                Wait Sleep waitTime=0.3
                Set DigitalOutput pin=config_out[1]; digitalValue=1
                Wait Sleep waitTime=0.3
                Loop Counting (count=2) loopVariable(name=Loop_80)
                  bajar := pose_add(get_actual_tcp_pose(), bajada_broca)
                  Waypoint Waypoint (Variable): motionParameters(jointSpeed=1.047198 jointAcceleration=1.396263 cartesianSpeed=0.001 cartesianAcceleration=0.005); variable=bajar
                  subir := pose_sub(get_actual_tcp_pose(), bajada_broca)
                  Waypoint Waypoint (Variable): motionParameters(jointSpeed=1.047198 jointAcceleration=1.396263 cartesianSpeed=0.005 cartesianAcceleration=0.01); variable=subir
                  bajada_broca := pose_sub(bajada_broca, bajada)
                MoveDirectionNode (selectedDirection=ZPlus toolParams=0.03, 0.035)
                  Until DISTANCE (allowActions=false deceleration=3 distanceNodeType=STOP) Distance=0.06; motionParameters(blendRadius=0)
                Set DigitalOutput pin=config_out[1]; digitalValue=0
                barreno_actual := barreno_actual+1
                If barreno_actual>barrenos_menos1
                  cambiar_broca := True
                SuppressedNode
                  Call Quitar_broca
                SuppressedNode
                  Call Poner_broca
      Popup Message (haltProgram=false message=Linea2 con chica Terminada! inputType=Text)
    Folder Broca_3
      Folder Linea3
        Folder Marcar_puntos
          MoveL speed 100 mm/s, acceleration 500 mm/s^2 (useActiveTCP=true) feature=Base
            Waypoint punto_inicio1: TCP in base x=646.451 y=-11.704 z=260.166 mm, rx=2.1511 ry=2.2897 rz=0 rad; joints [-205.616, -96.356, 115.768, -18.693, -308.324, -0.329] deg; TCP offset x=0.411 y=-218.298 z=37.994 mm, rx=1.558 ry=-0.1255 rz=0.1212 rad
            Waypoint Linea3_A: TCP in base x=460.55 y=-395.563 z=80.682 mm, rx=3.1326 ry=-0.0943 rz=0.0057 rad; joints [-228.865, -86.051, 126.783, -40.72, -234.593, 0.309] deg; TCP offset x=0.411 y=-218.298 z=37.994 mm, rx=1.558 ry=-0.1255 rz=0.1212 rad
            Waypoint Linea3_B: TCP in base x=664.301 y=-395.445 z=81.308 mm, rx=3.1326 ry=-0.0943 rz=0.0057 rad; joints [-215.162, -70.126, 106.29, -36.16, -220.885, 0.318] deg
            Waypoint Linea3_C: TCP in base x=689.223 y=-395.791 z=80.699 mm, rx=3.1326 ry=-0.0943 rz=0.0057 rad; joints [-213.996, -68.184, 103.511, -35.323, -219.718, 0.318] deg
            Waypoint Linea3_D: TCP in base x=892.727 y=-396.221 z=80.325 mm, rx=3.1326 ry=-0.0943 rz=0.0057 rad; joints [-206.597, -52.057, 77.467, -25.419, -212.299, 0.312] deg
            Waypoint Linea3_E: TCP in base x=918.375 y=-396.594 z=80.115 mm, rx=3.1326 ry=-0.0943 rz=0.0057 rad; joints [-205.9, -49.825, 73.601, -23.787, -211.599, 0.31] deg
            Waypoint Linea3_F: TCP in base x=1146.287 y=-396.633 z=80.258 mm, rx=3.1324 ry=-0.0938 rz=0.0063 rad; joints [-200.88, -21.042, 19.258, 1.725, -206.53, 0.288] deg; TCP offset x=0.411 y=-218.298 z=37.994 mm, rx=1.558 ry=-0.1255 rz=0.1212 rad
        Folder AB
          'desbaste_inicial'
          bajada_broca := p[0,0,-0.012,0,0,0]
          barrenos_menos1 := 8
          barreno_actual := 0
          Loop While (checkContinuously=false) expression=barreno_actual≤barrenos_menos1
            Folder Perforacion
              MoveL speed 100 mm/s, acceleration 500 mm/s^2 (useActiveTCP=true) feature=Base
                internos := interpolate_pose(Linea3_A, Linea3_B, barreno_actual/barrenos_menos1)
                Waypoint Waypoint (Variable): variable=internos
                'desbaste_inicial'
                bajada_broca := p[0,0,-0.012,0,0,0]
                bajada := p[0,0,0.012,0,0,0]
                MoveDirectionNode (selectedDirection=ZMinus toolParams=0.02, 0.015)
                  Until DISTANCE (allowActions=false deceleration=3 distanceNodeType=STOP) Distance=0.06; motionParameters(blendRadius=0)
                Popup Message (haltProgram=false message=punto contacto alanzdo inputType=Text)
                MoveDirectionNode (selectedDirection=ZPlus toolParams=0.003, 0.005)
                  Until DISTANCE (allowActions=false deceleration=3 distanceNodeType=STOP) Distance=0.002; motionParameters(blendRadius=0)
                Wait Sleep waitTime=0.3
                Set DigitalOutput pin=config_out[1]; digitalValue=1
                Wait Sleep waitTime=0.3
                Loop Counting (count=2) loopVariable(name=Loop_82)
                  bajar := pose_add(get_actual_tcp_pose(), bajada_broca)
                  Waypoint Waypoint (Variable): motionParameters(jointSpeed=1.047198 jointAcceleration=1.396263 cartesianSpeed=0.001 cartesianAcceleration=0.005); variable=bajar
                  subir := pose_sub(get_actual_tcp_pose(), bajada_broca)
                  Waypoint Waypoint (Variable): motionParameters(jointSpeed=1.047198 jointAcceleration=1.396263 cartesianSpeed=0.01 cartesianAcceleration=0.01); variable=subir
                  bajada_broca := pose_sub(bajada_broca, bajada)
                MoveDirectionNode (selectedDirection=ZPlus toolParams=0.03, 0.035)
                  Until DISTANCE (allowActions=false deceleration=3 distanceNodeType=STOP) Distance=0.06; motionParameters(blendRadius=0)
                Set DigitalOutput pin=config_out[1]; digitalValue=0
                barreno_actual := barreno_actual+1
                SuppressedNode
                  Call Quitar_broca
                SuppressedNode
                  Call Poner_broca
        Folder CD
          'desbaste_inicial'
          bajada_broca := p[0,0,-0.012,0,0,0]
          barrenos_menos1 := 8
          barreno_actual := 0
          Loop While (checkContinuously=false) expression=barreno_actual≤barrenos_menos1
            Folder Perforacion
              MoveL speed 100 mm/s, acceleration 500 mm/s^2 (useActiveTCP=true) feature=Base
                internos := interpolate_pose(Linea3_C, Linea3_D, barreno_actual/barrenos_menos1)
                Waypoint Waypoint (Variable): variable=internos
                'desbaste_inicial'
                bajada_broca := p[0,0,-0.012,0,0,0]
                bajada := p[0,0,0.012,0,0,0]
                MoveDirectionNode (selectedDirection=ZMinus toolParams=0.015, 0.02)
                  Until DISTANCE (allowActions=false deceleration=3 distanceNodeType=STOP) Distance=0.06; motionParameters(blendRadius=0)
                Popup Message (haltProgram=false message=punto contacto alanzdo inputType=Text)
                MoveDirectionNode (selectedDirection=ZPlus toolParams=0.003, 0.005)
                  Until DISTANCE (allowActions=false deceleration=3 distanceNodeType=STOP) Distance=0.002; motionParameters(blendRadius=0)
                Wait Sleep waitTime=0.3
                Set DigitalOutput pin=config_out[1]; digitalValue=1
                Wait Sleep waitTime=0.3
                Loop Counting (count=2) loopVariable(name=Loop_84)
                  bajar := pose_add(get_actual_tcp_pose(), bajada_broca)
                  Waypoint Waypoint (Variable): motionParameters(jointSpeed=1.047198 jointAcceleration=1.396263 cartesianSpeed=0.001 cartesianAcceleration=0.005); variable=bajar
                  subir := pose_sub(get_actual_tcp_pose(), bajada_broca)
                  Waypoint Waypoint (Variable): motionParameters(jointSpeed=1.047198 jointAcceleration=1.396263 cartesianSpeed=0.01 cartesianAcceleration=0.01); variable=subir
                  bajada_broca := pose_sub(bajada_broca, bajada)
                MoveDirectionNode (selectedDirection=ZPlus toolParams=0.03, 0.035)
                  Until DISTANCE (allowActions=false deceleration=3 distanceNodeType=STOP) Distance=0.06; motionParameters(blendRadius=0)
                Set DigitalOutput pin=config_out[1]; digitalValue=0
                barreno_actual := barreno_actual+1
                SuppressedNode
                  Call Quitar_broca
                SuppressedNode
                  Call Poner_broca
        Folder EF
          'desbaste_inicial'
          bajada_broca := p[0,0,-0.012,0,0,0]
          barrenos_menos1 := 9
          barreno_actual := 0
          Loop While (checkContinuously=false) expression=barreno_actual≤barrenos_menos1
            Folder Perforacion
              MoveL speed 100 mm/s, acceleration 500 mm/s^2 (useActiveTCP=true) feature=Base
                internos := interpolate_pose(Linea3_E, Linea3_F, barreno_actual/barrenos_menos1)
                Waypoint Waypoint (Variable): variable=internos
                'desbaste_inicial'
                bajada_broca := p[0,0,-0.012,0,0,0]
                bajada := p[0,0,0.012,0,0,0]
                MoveDirectionNode (selectedDirection=ZMinus toolParams=0.02, 0.015)
                  Until DISTANCE (allowActions=false deceleration=3 distanceNodeType=STOP) Distance=0.06; motionParameters(blendRadius=0)
                Popup Message (haltProgram=false message=punto contacto alanzdo inputType=Text)
                MoveDirectionNode (selectedDirection=ZPlus toolParams=0.003, 0.005)
                  Until DISTANCE (allowActions=false deceleration=3 distanceNodeType=STOP) Distance=0.002; motionParameters(blendRadius=0)
                Wait Sleep waitTime=0.3
                Set DigitalOutput pin=config_out[1]; digitalValue=1
                Wait Sleep waitTime=0.3
                Loop Counting (count=2) loopVariable(name=Loop_86)
                  bajar := pose_add(get_actual_tcp_pose(), bajada_broca)
                  Waypoint Waypoint (Variable): motionParameters(jointSpeed=1.047198 jointAcceleration=1.396263 cartesianSpeed=0.001 cartesianAcceleration=0.005); variable=bajar
                  subir := pose_sub(get_actual_tcp_pose(), bajada_broca)
                  Waypoint Waypoint (Variable): motionParameters(jointSpeed=1.047198 jointAcceleration=1.396263 cartesianSpeed=0.01 cartesianAcceleration=0.01); variable=subir
                  bajada_broca := pose_sub(bajada_broca, bajada)
                MoveDirectionNode (selectedDirection=ZPlus toolParams=0.03, 0.035)
                  Until DISTANCE (allowActions=false deceleration=3 distanceNodeType=STOP) Distance=0.06; motionParameters(blendRadius=0)
                Set DigitalOutput pin=config_out[1]; digitalValue=0
                barreno_actual := barreno_actual+1
                SuppressedNode
